// TIA Portal V20 export
DATA_BLOCK "ControlNodes"   // DB82
{ DB_Accessible_From_OPC_UA := 'FALSE' }
AUTHOR : ERsystem_FA2_DH. Kim
// stored: DBAccessibleFromOPCUA false, DBAccessibleFromWebserver false, MemoryReserve 100, Namespace Unit1.Em5
   VAR
      em { ExternalWritable := 'False'} : "LAF_typeEmControlNode";
      cm : Struct
         Interlock : Struct
            cathodeMainPnP1AxisX : "LER_typeAxisInterlock";
            cathodeMainPnP2AxisX : "LER_typeAxisInterlock";
            cathodeMainPnP1AxisY : "LER_typeAxisInterlock";
            cathodeMainPnP1AxisZ : "LER_typeAxisInterlock";
            cathodeMainPnP2AxisZ : "LER_typeAxisInterlock";
            cathodeAlignTableAxisX : "LER_typeAxisInterlock";
            cathodeAlignTableAxisY1 : "LER_typeAxisInterlock";
            cathodeAlignTableAxisY2 : "LER_typeAxisInterlock";
            cathodeMainPnP1RotaryCwCcw : "LER_typeTwoWayActInterlock";
            cathodeMainPnP1SuctionPlateVacuum : "LER_typeTwoWayActInterlock";
            cathodeMainPnP2SuctionPlateVacuum : "LER_typeTwoWayActInterlock";
            cathodeAlignTableSuctionPlateVacuum : "LER_typeTwoWayActInterlock";
            cathodeGlassCleaning : "LER_typeTwoWayActInterlock";
            cathodeNgPnpUpDown : "LER_typeTwoWayActInterlock";
            cathodeNgPnp1stFwdBwd : "LER_typeTwoWayActInterlock";
            cathodeNgPnp2ndFwdBwd : "LER_typeTwoWayActInterlock";
            cathodeMaintenanceMovingFixFwdBwd : "LER_typeTwoWayActInterlock";
            cathodeNgBoxLiftUpDown : "LER_typeTwoWayActInterlock";
            cathodeNgBoxLockUpDown : "LER_typeTwoWayActInterlock";
            cathodeNgPnpVaccum : "LER_typeTwoWayActInterlock";
            cathodeConveyorCoverFwdBwd : "LER_typeTwoWayActInterlock";
            cathodeConveyorPickUpBlower : "LER_typeTwoWayActInterlock";
         END_STRUCT;
         axisCommand : Struct
            cathodeMainPnP1AxisX : "LER_typeAxisCommand";
            cathodeMainPnP2AxisX : "LER_typeAxisCommand";
            cathodeMainPnP1AxisY : "LER_typeAxisCommand";
            cathodeMainPnP1AxisZ : "LER_typeAxisCommand";
            cathodeMainPnP2AxisZ : "LER_typeAxisCommand";
            cathodeAlignTableAxisX : "LER_typeAxisCommand";
            cathodeAlignTableAxisY1 : "LER_typeAxisCommand";
            cathodeAlignTableAxisY2 : "LER_typeAxisCommand";
         END_STRUCT;
         softCam : "Unit1.type_emRelations_em5_SoftCam";
         brakeTest : Struct
            cathodeMainPnP1AxisZ : "LER_typeBrakeTestEmControlNoeds";
            cathodeMainPnP2AxisZ : "LER_typeBrakeTestEmControlNoeds";
         END_STRUCT;
      END_STRUCT;
      mainPnP : Struct
         jobs : "LAF_typeJobs";
         sequence { S7_SetPoint := 'True'} : "LAF_typeSequence";
         "step" { S7_SetPoint := 'True'} : "LER_typeStep";
         jobInterface : Struct
            homeJob10 : "LER_typeJobInterface";
            homeJob1 : "LER_typeJobInterface";
            loadJob2 : "LER_typeJobInterface";
            unloadJob3 : "LER_typeJobInterface";
            avoidJob4 : "LER_typeJobInterface";
            oneLoadJob5 : "LER_typeJobInterface";
            oneUnLoadJob6 : "LER_typeJobInterface";
         END_STRUCT;
         preOperationCheck : Struct
            partNoDetect1 : Bool;   // MainPnP1/2 No Have Cell In LoadPos
            partNoDetect2 : Bool;
            partDetect1 : Bool;
            partDetect2 : Bool;
            partNG : Bool;
            Bool6 : Bool;
            Bool7 : Bool;
            Bool8 : Bool;   // MainPnP1 Have Cell
            Bool9 : Bool;   // MainPnP1/2 No Have Cell In UnLoadPos
            Bool10 : Bool;   // MainPnP1/2 Have Cell
            Bool11 : Bool;   // MainPnP1/2 Have Cell But Cathde Turn
            Bool12 : Bool;   // EM5 Ready For Motion
            Bool13 : Bool;
            Bool14 : Bool;
            Bool15 : Bool;
            Bool16 : Bool;
            Bool17 : Bool;
            Bool18 : Bool;
            Bool19 : Bool;
            Bool20 : Bool;
         END_STRUCT;
      END_STRUCT;
      alignTable : Struct
         jobs : "LAF_typeJobs";
         sequence { S7_SetPoint := 'True'} : "LAF_typeSequence";
         "step" { S7_SetPoint := 'True'} : "LER_typeStep";
         jobInterface : Struct
            homeJob1 : "LER_typeJobInterface";
            loadJob2 : "LER_typeJobInterface";
            visionJob3 : "LER_typeJobInterface";
            unloadJob4 : "LER_typeJobInterface";
         END_STRUCT;
         preOperationCheck : Struct
            partNoDetect1 : Bool;   // AlignTable No Have Cell In WaitPos
            partNoDetect2 : Bool;   // AlignTable No Have Cell In AdjustPos
            partDetect1 : Bool;   // AlignTable Have Cell In WaitPos
            partDetect2 : Bool;   // AlignTable Have Cell In AdjustPos
            Bool5 : Bool;
            Bool6 : Bool;
            Bool7 : Bool;
            Bool8 : Bool;
            Bool9 : Bool;
            Bool10 : Bool;
            Bool11 : Bool;
            Bool12 : Bool;
            Bool13 : Bool;
            Bool14 : Bool;
            Bool15 : Bool;
            Bool16 : Bool;
            Bool17 : Bool;
            Bool18 : Bool;
            Bool19 : Bool;
            Bool20 : Bool;
         END_STRUCT;
      END_STRUCT;
      ngPnP : Struct
         jobs : "LAF_typeJobs";
         sequence { S7_SetPoint := 'True'} : "LAF_typeSequence";
         "step" { S7_SetPoint := 'True'} : "LER_typeStep";
         jobInterface : Struct
            homeJob1 : "LER_typeJobInterface";
            loadJob2 : "LER_typeJobInterface";
            unloadJob3 : "LER_typeJobInterface";
         END_STRUCT;
         preOperationCheck : Struct
            partNoDetect : Bool;
            partDetect : Bool;
            Bool3 : Bool;
            Bool4 : Bool;
            Bool5 : Bool;
            Bool6 : Bool;
            Bool7 : Bool;
            Bool8 : Bool;
            Bool9 : Bool;
            Bool10 : Bool;
            Bool11 : Bool;
            Bool12 : Bool;
            Bool13 : Bool;
            Bool14 : Bool;
            Bool15 : Bool;
            Bool16 : Bool;
            Bool17 : Bool;
            Bool18 : Bool;
            Bool19 : Bool;
            Bool20 : Bool;
         END_STRUCT;
      END_STRUCT;
      gaugeRnR : Struct
         jobs : "LAF_typeJobs";
         sequence { S7_SetPoint := 'True'} : "LAF_typeSequence";
         "step" { S7_SetPoint := 'True'} : "LER_typeStep";
         jobInterface : Struct
            commonReadyJob1 : "LER_typeJobInterface";
            commonGetMasterPieceJob2 { S7_SetPoint := 'True'} : "LER_typeJobInterface";
            "1StackMainPnP2ToStackTableJob19" { S7_SetPoint := 'True'} : "LER_typeJobInterface";
            "1StackStackTableToMainPnP2Job20" { S7_SetPoint := 'True'} : "LER_typeJobInterface";
         END_STRUCT;
         homeCheck : Struct
            home : Bool;
         END_STRUCT;
      END_STRUCT;
      ReelCutInterface : Struct
         readyMasterPiece : Bool;
      END_STRUCT;
      emRelations : Struct
         em6 : Struct
            reqStackTableVaccum : Bool;
            reqStackTableBlow : Bool;
            readyGaugeRnR : Bool;
            doneStackTableVaccum : Bool;
            doneStackTableBlow : Bool;
            doneGaugeRnR : Bool;
            softCam : "Unit1.type_emRelations_em6_SoftCam";
         END_STRUCT;
      END_STRUCT;
      cmPnp1stCathodeDetect { S7_SetPoint := 'True'} : "LBC_typeDigitalSignalControlNode";
      cmPnp2ndCathodeDetect { S7_SetPoint := 'True'} : "LBC_typeDigitalSignalControlNode";
      cmCathodeAlignTableElectrodeDetect { S7_SetPoint := 'True'} : "LBC_typeDigitalSignalControlNode";
      cmCathodeNgPnpElectrodeDetect { S7_SetPoint := 'True'} : "LBC_typeDigitalSignalControlNode";
      cmCathodeNgBoxFullSensorDetect { S7_SetPoint := 'True'} : "LBC_typeDigitalSignalControlNode";
      cmCathodeNgBoxDetect { S7_SetPoint := 'True'} : "LBC_typeDigitalSignalControlNode";
      cmCathodeMainPnP1AxisX { ExternalAccessible := 'False'; ExternalVisible := 'False'; ExternalWritable := 'False'} : "LBC_typeAxis64PosControlNode";
      cmCathodeMainPnP2AxisX { ExternalAccessible := 'False'; ExternalVisible := 'False'; ExternalWritable := 'False'} : "LBC_typeAxis64PosControlNode";
      cmCathodeMainPnP1AxisY { ExternalAccessible := 'False'; ExternalVisible := 'False'; ExternalWritable := 'False'} : "LBC_typeAxis64PosControlNode";
      cmCathodeMainPnP1AxisZ { ExternalAccessible := 'False'; ExternalVisible := 'False'; ExternalWritable := 'False'} : "LBC_typeAxis64PosControlNode";
      cmCathodeMainPnP2AxisZ { ExternalAccessible := 'False'; ExternalVisible := 'False'; ExternalWritable := 'False'} : "LBC_typeAxis64PosControlNode";
      cmCathodeAlignTableAxisX { ExternalAccessible := 'False'; ExternalVisible := 'False'; ExternalWritable := 'False'} : "LBC_typeAxis64PosControlNode";
      cmCathodeAlignTableAxisY1 { ExternalAccessible := 'False'; ExternalVisible := 'False'; ExternalWritable := 'False'} : "LBC_typeAxis64PosControlNode";
      cmCathodeAlignTableAxisY2 { ExternalAccessible := 'False'; ExternalVisible := 'False'; ExternalWritable := 'False'} : "LBC_typeAxis64PosControlNode";
      cmCathodeMainPnP1RotaryCwCcw { ExternalAccessible := 'False'; ExternalVisible := 'False'; ExternalWritable := 'False'} : "LBC_typeTwoWayActuatorControlNode";
      cmCathodeMainPnP1SuctionPlateVacuum { ExternalAccessible := 'False'; ExternalVisible := 'False'; ExternalWritable := 'False'} : "LBC_typeTwoWayActuatorControlNode";
      cmCathodeMainPnP2SuctionPlateVacuum { ExternalAccessible := 'False'; ExternalVisible := 'False'; ExternalWritable := 'False'} : "LBC_typeTwoWayActuatorControlNode";
      cmCathodeAlignTableSuctionPlateVacuum { ExternalAccessible := 'False'; ExternalVisible := 'False'; ExternalWritable := 'False'} : "LBC_typeTwoWayActuatorControlNode";
      cmCathodeGlassCleaning { ExternalAccessible := 'False'; ExternalVisible := 'False'; ExternalWritable := 'False'} : "LBC_typeTwoWayActuatorControlNode";
      cmCathodeNgPnpUpDown { ExternalAccessible := 'False'; ExternalVisible := 'False'; ExternalWritable := 'False'} : "LBC_typeTwoWayActuatorControlNode";
      cmCathodeNgPnp1stFwdBwd { ExternalAccessible := 'False'; ExternalVisible := 'False'; ExternalWritable := 'False'} : "LBC_typeTwoWayActuatorControlNode";
      cmCathodeNgPnp2ndFwdBwd { ExternalAccessible := 'False'; ExternalVisible := 'False'; ExternalWritable := 'False'; S7_SetPoint := 'True'} : "LBC_typeTwoWayActuatorControlNode";
      cmCathodeMaintenanceMovingFixFwdBwd { ExternalAccessible := 'False'; ExternalVisible := 'False'; ExternalWritable := 'False'} : "LBC_typeTwoWayActuatorControlNode";
      cmCathodeNgBoxLiftUpDown { ExternalAccessible := 'False'; ExternalVisible := 'False'; ExternalWritable := 'False'; S7_SetPoint := 'True'} : "LBC_typeTwoWayActuatorControlNode";
      cmCathodeNgBoxLockUpDown { ExternalAccessible := 'False'; ExternalVisible := 'False'; ExternalWritable := 'False'; S7_SetPoint := 'True'} : "LBC_typeTwoWayActuatorControlNode";
      cmCathodeNgPnpVaccum { ExternalAccessible := 'False'; ExternalVisible := 'False'; ExternalWritable := 'False'} : "LBC_typeTwoWayActuatorControlNode";
      cmCathodeConveyorCoverFwdBwd { S7_SetPoint := 'True'} : "LBC_typeTwoWayActuatorControlNode";
      cmCathodeConveyorPickUpBlower { S7_SetPoint := 'True'} : "LBC_typeTwoWayActuatorControlNode";
      cmCathodeVisionControllerInterface { ExternalAccessible := 'False'; ExternalVisible := 'False'; ExternalWritable := 'False'} : "LER_typeVisionControlNode";
   END_VAR
BEGIN
   em.commands.enable := FALSE;
   em.commands.acknowledge := FALSE;
   em.commands.disableAlarms := FALSE;
   em.commands.activateSimulation := FALSE;
   em.commands.home := FALSE;
   em.commands.moveToInitialPosition := FALSE;
   em.commands.directModeControl.current := 2;
   em.commands.directModeControl.production := FALSE;
   em.commands.directModeControl.maintenance := TRUE;
   em.commands.directModeControl.manual := FALSE;
   em.commands.directModeControl.nomode := FALSE;
   em.commands.directModeControl.sleep := FALSE;
   em.commands.directModeControl.deepsleep := FALSE;
   em.commands.directModeControl.userMode04 := FALSE;
   em.commands.directModeControl.userMode05 := FALSE;
   em.commands.directModeControl.userMode06 := FALSE;
   em.commands.directModeControl.userMode07 := FALSE;
   em.commands.directModeControl.userMode08 := FALSE;
   em.commands.directModeControl.userMode09 := FALSE;
   em.commands.directModeControl.userMode10 := FALSE;
   em.commands.directModeControl.userMode11 := FALSE;
   em.commands.directModeControl.userMode12 := FALSE;
   em.commands.directModeControl.userMode13 := FALSE;
   em.commands.directStateControl.current := 2;
   em.commands.directStateControl.clearing := FALSE;
   em.commands.directStateControl.stopped := TRUE;
   em.commands.directStateControl.starting := FALSE;
   em.commands.directStateControl.idle := FALSE;
   em.commands.directStateControl.suspended := FALSE;
   em.commands.directStateControl.execute := FALSE;
   em.commands.directStateControl.stopping := FALSE;
   em.commands.directStateControl.aborting := FALSE;
   em.commands.directStateControl.aborted := FALSE;
   em.commands.directStateControl.holding := FALSE;
   em.commands.directStateControl.held := FALSE;
   em.commands.directStateControl.unholding := FALSE;
   em.commands.directStateControl.suspending := FALSE;
   em.commands.directStateControl.unsuspending := FALSE;
   em.commands.directStateControl.resetting := FALSE;
   em.commands.directStateControl.completing := FALSE;
   em.commands.directStateControl.complete := FALSE;
   em.status.enabled := FALSE;
   em.status.acknowledgeActive := FALSE;
   em.status.alarmsDisabled := FALSE;
   em.status.simulationActive := FALSE;
   em.status.safetyReleased := TRUE;
   em.status.initialized := FALSE;
   em.status.homed := TRUE;
   em.status.safeState := FALSE;
   em.status.stateComplete := TRUE;
   // mainPnP."step".action1[101] : Step[101] : JOB[1] Condition
   // mainPnP."step".action1[110] : Step[110] : Main P&P 1,2 Z-Axis Wait Pos
   // mainPnP."step".action1[111] : Step[111] : Main P&P 1 Y-Axis Wait Pos
   // mainPnP."step".action1[112] : Step[112] : Main P&P 1,2 X-Axis Wait(=Load) Pos
   // mainPnP."step".action1[113] : Step[113] : Main P&P 1 Rotary Cylinder InHomePos(=Clock Wise)
   // mainPnP."step".action1[114] : Step[114] : Main P&P 1 Z-Axis Load Pos
   // mainPnP."step".action1[115] : Step[115] : Main P&P 1 Vaccum On
   // mainPnP."step".action1[116] : Step[116] : Main P&P 1 Pick Up Blow On
   // mainPnP."step".action1[117] : Step[117] : Main P&P 1,2 Z-Axis Wait Pos
   // mainPnP."step".action1[120] : Step[120] : Main P&P 1,2 X-Axis Unload Pos
   // mainPnP."step".action1[121] : Step[121] : Main P&P 1 Rotary Cylinder InWorkPos(=Counter Clock Wise)
   // mainPnP."step".action1[122] : Step[122] : Main P&P 1 Z-Axis Unload Pos [Request Check]
   // mainPnP."step".action1[123] : Step[123] : Main P&P → Align Table [Vacuum On Request]
   // mainPnP."step".action1[124] : Step[124] : Main P&P 1 Vaccum Off
   // mainPnP."step".action1[125] : Step[125] : Main P&P 1,2 Z-Axis Wait Pos
   // mainPnP."step".action1[130] : Step[130] : Main P&P 1,2 X-Axis Load Pos
   // mainPnP."step".action1[131] : Step[131] : Main P&P 1 Rotary Cylinder InHomePos(=Clock Wise)
   // mainPnP."step".action1[132] : Step[132] : Main P&P 1,2 Z-Axis Load Pos [Request Check]
   // mainPnP."step".action1[133] : Step[133] : Main P&P 1,2 Vaccum On
   // mainPnP."step".action1[134] : Step[134] : Main P&P → Align Table [Vacuum Off Request] / Pick Up Blow On
   // mainPnP."step".action1[135] : Step[135] : Main P&P 1,2 Z-Axis Wait Pos
   // mainPnP."step".action1[140] : Step[140] : Main P&P 1,2 X-Axis Unload Pos
   // mainPnP."step".action1[141] : Step[141] : Main P&P 1 Rotary Cylinder InWorkPos(=Counter Clock Wise)
   // mainPnP."step".action1[142] : Step[142] : Main P&P 1,2 Z-Axis Unload Pos [Request Check]
   // mainPnP."step".action1[143] : Step[143] : Main P&P → Align Table [Vacuum On Request] / Mendrel [Clamp Request]
   // mainPnP."step".action1[144] : Step[144] : Main P&P 1,2 Vaccum Off
   // mainPnP."step".action1[145] : Step[145] : Main P&P 1,2 Z-Axis Wait Pos
   // mainPnP."step".action1[180] : Step[180] : Main P&P 1,2 X-Axis Load Pos
   // mainPnP."step".action1[181] : Step[181] : Main P&P 1 Rotary Cylinder InHomePos(=Clock Wise)
   // mainPnP."step".action1[182] : Step[182] : Main P&P 1,2 Z-Axis Load Pos [Request Check]
   // mainPnP."step".action1[183] : Step[183] : Main P&P 1,2 Vaccum On
   // mainPnP."step".action1[184] : Step[184] : Main P&P → Align Table [Vacuum Off Request] / Pick Up Blow On
   // mainPnP."step".action1[185] : Step[185] : Main P&P 1,2 Z-Axis Avoid Pos
   // mainPnP."step".action1[190] : Step[190] : JOB[1] Step End
   // mainPnP."step".action1[201] : Step[201] : JOB[2] Condition
   // mainPnP."step".action1[210] : Step[210] : Main P&P 1,2 Z-Axis Wait Pos
   // mainPnP."step".action1[220] : Step[220] : Main P&P 1,2 X-Axis Load Pos
   // mainPnP."step".action1[230] : Step[230] : Main P&P 1 Rotary Cylinder InHomePos(=Clock Wise)
   // mainPnP."step".action1[240] : Step[240] : Main P&P 1.2 Z-Axis Load Pos
   // mainPnP."step".action1[250] : Step[250] : Main P&P 1,2 Vaccum On
   // mainPnP."step".action1[260] : Step[260] : Main P&P → Align Table [Vacuum Off Request] / Pick Up Blow On
   // mainPnP."step".action1[280] : Step[280] : Main P&P 1,2 Z-Axis Wait Pos
   // mainPnP."step".action1[290] : Step[290] : JOB[2] Condition
   // mainPnP."step".action1[301] : Step[301] : JOB[3] Condition
   // mainPnP."step".action1[310] : Step[310] : Main P&P 1,2 Z-Axis Wait Pos
   // mainPnP."step".action1[320] : Step[320] : Main P&P 1,2 X-Axis Unload Pos
   // mainPnP."step".action1[330] : Step[330] : Main P&P 1 Rotary Cylinder InWorkPos(=Counter Clock Wise)
   // mainPnP."step".action1[340] : Step[340] : Main P&P 1.2 Z-Axis Unload Pos
   // mainPnP."step".action1[350] : Step[350] : Main P&P → Align Table [Vacuum On Request] / Mendrel [Clamp Request]
   // mainPnP."step".action1[360] : Step[360] : Main P&P 1.2 Vaccum Off
   // mainPnP."step".action1[380] : Step[380] : Main P&P 1,2 Z-Axis Wait Pos
   // mainPnP."step".action1[390] : Step[390] : JOB[3] Condition
   // mainPnP."step".action1[401] : Step[401] : JOB[4] Condition
   // mainPnP."step".action1[420] : Step[420] : Main P&P 1 X-Axis Load Pos, Main P&P 2 X-Axis Unload Pos
   // mainPnP."step".action1[430] : Step[430] : Main P&P 1 Rotary Cylinder InHomePos(=Clock Wise)
   // mainPnP."step".action1[490] : Step[490] : JOB[3] Condition
   // mainPnP."step".transition1[101] : Step[101] : JOB[1] Condition
   // mainPnP."step".transition1[110] : Step[110] : Main P&P 1,2 Z-Axis Wait Pos
   // mainPnP."step".transition1[111] : Step[111] : Main P&P 1 Y-Axis Wait Pos
   // mainPnP."step".transition1[112] : Step[112] : Main P&P 1,2 X-Axis Wait(=Load) Pos
   // mainPnP."step".transition1[113] : Step[113] : Main P&P 1 Rotary Cylinder InHomePos(=Clock Wise)
   // mainPnP."step".transition1[114] : Step[114] : Main P&P 1 Z-Axis Load Pos
   // mainPnP."step".transition1[115] : Step[115] : Main P&P 1 Vaccum On
   // mainPnP."step".transition1[116] : Step[116] : Main P&P 1 Pick Up Blow On
   // mainPnP."step".transition1[117] : Step[117] : Main P&P 1,2 Z-Axis Wait Pos
   // mainPnP."step".transition1[120] : Step[120] : Main P&P 1,2 X-Axis Unload Pos
   // mainPnP."step".transition1[121] : Step[121] : Main P&P 1 Rotary Cylinder InWorkPos(=Counter Clock Wise)
   // mainPnP."step".transition1[122] : Step[122] : Main P&P 1 Z-Axis Unload Pos [Request Check]
   // mainPnP."step".transition1[123] : Step[123] : Main P&P → Align Table [Vacuum On Request]
   // mainPnP."step".transition1[124] : Step[124] : Main P&P 1 Vaccum Off
   // mainPnP."step".transition1[125] : Step[125] : Main P&P 1,2 Z-Axis Wait Pos
   // mainPnP."step".transition1[130] : Step[130] : Main P&P 1,2 X-Axis Load Pos
   // mainPnP."step".transition1[131] : Step[131] : Main P&P 1 Rotary Cylinder InHomePos(=Clock Wise)
   // mainPnP."step".transition1[132] : Step[132] : Main P&P 1,2 Z-Axis Load Pos [Request Check]
   // mainPnP."step".transition1[133] : Step[133] : Main P&P 1,2 Vaccum On
   // mainPnP."step".transition1[134] : Step[134] : Main P&P → Align Table [Vacuum Off Request] / Pick Up Blow On
   // mainPnP."step".transition1[135] : Step[135] : Main P&P 1,2 Z-Axis Wait Pos
   // mainPnP."step".transition1[140] : Step[140] : Main P&P 1,2 X-Axis Unload Pos
   // mainPnP."step".transition1[141] : Step[141] : Main P&P 1 Rotary Cylinder InWorkPos(=Counter Clock Wise)
   // mainPnP."step".transition1[142] : Step[142] : Main P&P 1,2 Z-Axis Unload Pos [Request Check]
   // mainPnP."step".transition1[143] : Step[143] : Main P&P → Align Table [Vacuum On Request] / Mendrel [Clamp Request]
   // mainPnP."step".transition1[144] : Step[144] : Main P&P 1,2 Vaccum Off
   // mainPnP."step".transition1[145] : Step[145] : Main P&P 1,2 Z-Axis Wait Pos
   // mainPnP."step".transition1[180] : Step[180] : Main P&P 1,2 X-Axis Load Pos
   // mainPnP."step".transition1[181] : Step[181] : Main P&P 1 Rotary Cylinder InHomePos(=Clock Wise)
   // mainPnP."step".transition1[182] : Step[182] : Main P&P 1,2 Z-Axis Load Pos [Request Check]
   // mainPnP."step".transition1[183] : Step[183] : Main P&P 1,2 Vaccum On
   // mainPnP."step".transition1[184] : Step[184] : Main P&P → Align Table [Vacuum Off Request] / Pick Up Blow On
   // mainPnP."step".transition1[185] : Step[185] : Main P&P 1,2 Z-Axis Avoid Pos
   // mainPnP."step".transition1[190] : Step[190] : JOB[1] Step End
   // mainPnP."step".transition1[201] : Step[201] : JOB[2] Condition
   // mainPnP."step".transition1[210] : Step[210] : Main P&P 1,2 Z-Axis Wait Pos
   // mainPnP."step".transition1[220] : Step[220] : Main P&P 1,2 X-Axis Load Pos
   // mainPnP."step".transition1[230] : Step[230] : Main P&P 1 Rotary Cylinder InHomePos(=Clock Wise)
   // mainPnP."step".transition1[240] : Step[240] : Main P&P 1.2 Z-Axis Load Pos
   // mainPnP."step".transition1[250] : Step[250] : Main P&P 1,2 Vaccum On
   // mainPnP."step".transition1[260] : Step[260] : Main P&P → Align Table [Vacuum Off Request] / Pick Up Blow On
   // mainPnP."step".transition1[280] : Step[280] : Main P&P 1,2 Z-Axis Wait Pos
   // mainPnP."step".transition1[290] : Step[290] : JOB[2] Condition
   // mainPnP."step".transition1[301] : Step[301] : JOB[3] Condition
   // mainPnP."step".transition1[310] : Step[310] : Main P&P 1,2 Z-Axis Wait Pos
   // mainPnP."step".transition1[320] : Step[320] : Main P&P 1,2 X-Axis Unload Pos
   // mainPnP."step".transition1[330] : Step[330] : Main P&P 1 Rotary Cylinder InWorkPos(=Counter Clock Wise)
   // mainPnP."step".transition1[340] : Step[340] : Main P&P 1.2 Z-Axis Unload Pos
   // mainPnP."step".transition1[350] : Step[350] : Main P&P → Align Table [Vacuum On Request] / Mendrel [Clamp Request]
   // mainPnP."step".transition1[360] : Step[360] : Main P&P 1.2 Vaccum Off
   // mainPnP."step".transition1[380] : Step[380] : Main P&P 1,2 Z-Axis Wait Pos
   // mainPnP."step".transition1[390] : Step[390] : JOB[3] Condition
   // mainPnP."step".transition1[401] : Step[401] : JOB[4] Condition
   // mainPnP."step".transition1[420] : Step[420] : Main P&P 1 X-Axis Load Pos, Main P&P 2 X-Axis Unload Pos
   // mainPnP."step".transition1[430] : Step[430] : Main P&P 1 Rotary Cylinder InHomePos(=Clock Wise)
   // mainPnP."step".transition1[490] : Step[490] : JOB[3] Condition
   // alignTable."step".action1[101] : Step[101] : JOB[1] Condition
   // alignTable."step".action1[110] : Step[110] : Vaccum Off
   // alignTable."step".action1[120] : Step[120] : Glass Cleaning On [Main P&P Working Done Check]
   // alignTable."step".action1[140] : Step[140] : Align Table → Main P&P [Load Request]
   // alignTable."step".action1[141] : Step[141] : Vaccum On
   // alignTable."step".action1[142] : Step[142] : Align Table → Main P&P [Load Done] / [Vision Unuse Check]
   // alignTable."step".action1[150] : Step[150] : Vision Start
   // alignTable."step".action1[151] : Step[151] : Vision Result
   // alignTable."step".action1[152] : Step[152] : Align Table X,Y1,Y2-Axis Work Pos
   // alignTable."step".action1[160] : Step[160] : Align Table → Main P&P/NG P&P [Unload Request]
   // alignTable."step".action1[161] : Step[161] : Vaccum Off
   // alignTable."step".action1[162] : Step[162] : Align Table → Main P&P [Unload Done]
   // alignTable."step".action1[163] : Step[163] : Glass Cleaning On [Main P&P Homing Job Complete Check]
   // alignTable."step".action1[180] : Step[180] : Align Table X,Y1,Y2-Axis Wait Pos
   // alignTable."step".action1[190] : Step[190] : JOB[1] Step End
   // alignTable."step".action1[201] : Step[201] : JOB[2] Condition
   // alignTable."step".action1[210] : Step[210] : Align Table → Main P&P [Load Request]
   // alignTable."step".action1[220] : Step[220] : Vaccum On
   // alignTable."step".action1[230] : Step[230] : Align Table → Main P&P [Load Done]
   // alignTable."step".action1[290] : Step[290] : JOB[2] Condition
   // alignTable."step".action1[301] : Step[301] : JOB[3] Condition
   // alignTable."step".action1[310] : Step[310] : Vision Start
   // alignTable."step".action1[320] : Step[320] : Vision Result
   // alignTable."step".action1[380] : Step[380] : Align Table X,Y1,Y2-Axis Work Pos
   // alignTable."step".action1[390] : Step[390] : JOB[3] Condition
   // alignTable."step".action1[401] : Step[401] : JOB[4] Condition
   // alignTable."step".action1[410] : Step[410] : Align Table → Main P&P/NG P&P [Unload Request]
   // alignTable."step".action1[420] : Step[420] : Vaccum Off
   // alignTable."step".action1[430] : Step[430] : Align Table → Main P&P [Unload Done]
   // alignTable."step".action1[431] : Step[431] : Glass Cleaning On
   // alignTable."step".action1[480] : Step[480] : Align Table X,Y1,Y2-Axis Wait Pos
   // alignTable."step".transition1[101] : Step[101] : JOB[1] Condition
   // alignTable."step".transition1[110] : Step[110] : Vaccum Off
   // alignTable."step".transition1[120] : Step[120] : Glass Cleaning On [Main P&P Working Done Check]
   // alignTable."step".transition1[140] : Step[140] : Align Table → Main P&P [Load Request]
   // alignTable."step".transition1[141] : Step[141] : Vaccum On
   // alignTable."step".transition1[142] : Step[142] : Align Table → Main P&P [Load Done] / [Vision Unuse Check]
   // alignTable."step".transition1[150] : Step[150] : Vision Start
   // alignTable."step".transition1[151] : Step[151] : Vision Result
   // alignTable."step".transition1[152] : Step[152] : Align Table X,Y1,Y2-Axis Work Pos
   // alignTable."step".transition1[160] : Step[160] : Align Table → Main P&P/NG P&P [Unload Request]
   // alignTable."step".transition1[161] : Step[161] : Vaccum Off
   // alignTable."step".transition1[162] : Step[162] : Align Table → Main P&P [Unload Done]
   // alignTable."step".transition1[163] : Step[163] : Glass Cleaning On [Main P&P Homing Job Complete Check]
   // alignTable."step".transition1[180] : Step[180] : Align Table X,Y1,Y2-Axis Wait Pos
   // alignTable."step".transition1[190] : Step[190] : JOB[1] Step End
   // alignTable."step".transition1[201] : Step[201] : JOB[2] Condition
   // alignTable."step".transition1[210] : Step[210] : Align Table → Main P&P [Load Request]
   // alignTable."step".transition1[220] : Step[220] : Vaccum On
   // alignTable."step".transition1[230] : Step[230] : Align Table → Main P&P [Load Done]
   // alignTable."step".transition1[290] : Step[290] : JOB[2] Condition
   // alignTable."step".transition1[301] : Step[301] : JOB[3] Condition
   // alignTable."step".transition1[310] : Step[310] : Vision Start
   // alignTable."step".transition1[320] : Step[320] : Vision Result
   // alignTable."step".transition1[380] : Step[380] : Align Table X,Y1,Y2-Axis Work Pos
   // alignTable."step".transition1[390] : Step[390] : JOB[3] Condition
   // alignTable."step".transition1[401] : Step[401] : JOB[4] Condition
   // alignTable."step".transition1[410] : Step[410] : Align Table → Main P&P/NG P&P [Unload Request]
   // alignTable."step".transition1[420] : Step[420] : Vaccum Off
   // alignTable."step".transition1[430] : Step[430] : Align Table → Main P&P [Unload Done]
   // alignTable."step".transition1[431] : Step[431] : Glass Cleaning On
   // alignTable."step".transition1[480] : Step[480] : Align Table X,Y1,Y2-Axis Wait Pos
   // ngPnP."step".action1[101] : Step[101] : JOB[1] Condition
   // ngPnP."step".action1[110] : Step[110] : Vaccum Off
   // ngPnP."step".action1[120] : Step[120] : NG P&P Up
   // ngPnP."step".action1[130] : Step[130] : NG P&P 1,2 Backward
   // ngPnP."step".action1[180] : Step[180] : Lift Down
   // ngPnP."step".action1[190] : Step[190] : JOB[1] Step End
   // ngPnP."step".action1[201] : Step[201] : JOB[2] Condition
   // ngPnP."step".action1[210] : Step[210] : NG P&P 1,2 Forward
   // ngPnP."step".action1[220] : Step[220] : NG P&P Down
   // ngPnP."step".action1[230] : Step[230] : Vaccum On
   // ngPnP."step".action1[231] : Step[231] : NG P&P → Align Table [Loading Ready]
   // ngPnP."step".action1[240] : Step[240] : NG P&P Up
   // ngPnP."step".action1[280] : Step[280] : NG P&P 1,2 Backward
   // ngPnP."step".action1[290] : Step[290] : JOB[2] Condition
   // ngPnP."step".action1[301] : Step[301] : JOB[3] Condition
   // ngPnP."step".action1[320] : Step[320] : NG P&P Down
   // ngPnP."step".action1[330] : Step[330] : Vaccum Off
   // ngPnP."step".action1[340] : Step[340] : NG P&P Up
   // ngPnP."step".action1[390] : Step[390] : JOB[3] Condition
   // ngPnP."step".transition1[101] : Step[101] : JOB[1] Condition
   // ngPnP."step".transition1[110] : Step[110] : Vaccum Off
   // ngPnP."step".transition1[120] : Step[120] : NG P&P Up
   // ngPnP."step".transition1[130] : Step[130] : NG P&P 1,2 Backward
   // ngPnP."step".transition1[180] : Step[180] : Lift Down
   // ngPnP."step".transition1[190] : Step[190] : JOB[1] Step End
   // ngPnP."step".transition1[201] : Step[201] : JOB[2] Condition
   // ngPnP."step".transition1[210] : Step[210] : NG P&P 1,2 Forward
   // ngPnP."step".transition1[220] : Step[220] : NG P&P Down
   // ngPnP."step".transition1[230] : Step[230] : Vaccum On
   // ngPnP."step".transition1[231] : Step[231] : NG P&P → Align Table [Loading Ready]
   // ngPnP."step".transition1[240] : Step[240] : NG P&P Up
   // ngPnP."step".transition1[280] : Step[280] : NG P&P 1,2 Backward
   // ngPnP."step".transition1[290] : Step[290] : JOB[2] Condition
   // ngPnP."step".transition1[301] : Step[301] : JOB[3] Condition
   // ngPnP."step".transition1[320] : Step[320] : NG P&P Down
   // ngPnP."step".transition1[330] : Step[330] : Vaccum Off
   // ngPnP."step".transition1[340] : Step[340] : NG P&P Up
   // ngPnP."step".transition1[390] : Step[390] : JOB[3] Condition
   // gaugeRnR."step".action1[101] : Step[101] : JOB[1] Condition
   // gaugeRnR."step".action1[110] : Step[110] : MainPnP 1 Vaccum Off
   // gaugeRnR."step".action1[120] : Step[120] : MainPnP 2 Vaccum Off
   // gaugeRnR."step".action1[130] : Step[130] : AlignTable Vaccum Off
   // gaugeRnR."step".action1[190] : Step[190] : Job[1] Step End
   // gaugeRnR."step".action1[201] : Step[201] : JOB[2] Condition
   // gaugeRnR."step".action1[210] : Step[210] : MainPnP1 Z-Axis Conveyor Down
   // gaugeRnR."step".action1[220] : Step[220] : MainPnP1 C/V Blow On
   // gaugeRnR."step".action1[230] : Step[230] : MainPnP1 Vaccum On
   // gaugeRnR."step".action1[240] : Step[240] : MainPnP1 C/V Blow Off
   // gaugeRnR."step".action1[250] : Step[250] : MainPnP1 Z-Axis Up
   // gaugeRnR."step".action1[290] : Step[290] : Job[2] Step End
   // gaugeRnR."step".action1[301] : Step[301] : JOB[3] Condition
   // gaugeRnR."step".action1[310] : Step[310] : MainPnP2 X-Axis Move StackTable
   // gaugeRnR."step".action1[320] : Step[320] : MainPnP1 X-Axis Move AlignTable
   // gaugeRnR."step".action1[390] : Step[390] : Job[3] Step End
   // gaugeRnR."step".action1[401] : Step[401] : Job[4] Condtion
   // gaugeRnR."step".action1[410] : Step[410] : MainPnP1 Z-Axis Down AlginTable
   // gaugeRnR."step".action1[420] : Step[420] : MainPnP1 1 Vaccum Off
   // gaugeRnR."step".action1[430] : Step[430] : AlignTable Vaccum On
   // gaugeRnR."step".action1[440] : Step[440] : MainPnP 1 Z-Axis Up
   // gaugeRnR."step".action1[490] : Step[490] : Job[4] Step End
   // gaugeRnR."step".action1[501] : Step[501] : Job[5] Condtion
   // gaugeRnR."step".action1[510] : Step[510] : MainPnP1 X-Axis Move ReelCut Convyeor
   // gaugeRnR."step".action1[520] : Step[520] : MainPnP2 X-Axis Move AlignTable
   // gaugeRnR."step".action1[590] : Step[590] : Job[5] Step End
   // gaugeRnR."step".action1[601] : Step[601] : Job[6] Condtion
   // gaugeRnR."step".action1[610] : Step[610] : AlignTable Vision Trigger On
   // gaugeRnR."step".action1[620] : Step[620] : AlignTable Move Adjust Pos
   // gaugeRnR."step".action1[690] : Step[690] : Job[6] Step End
   // gaugeRnR."step".action1[701] : Step[701] : Job[7] Condtion
   // gaugeRnR."step".action1[710] : Step[710] : MainPnP2 Z-Axis Down AlignTagble
   // gaugeRnR."step".action1[720] : Step[720] : AlignTable Vaccum Off
   // gaugeRnR."step".action1[730] : Step[730] : MainPnP2 Vaccum On
   // gaugeRnR."step".action1[740] : Step[740] : MainPnP2 Z-Axis Up
   // gaugeRnR."step".action1[790] : Step[790] : Job[7] Step End
   // gaugeRnR."step".action1[801] : Step[801] : Job[8] Condtion
   // gaugeRnR."step".action1[810] : Step[810] : AlignTable Move Wait
   // gaugeRnR."step".action1[890] : Step[890] : Job[8] Step End
   // gaugeRnR."step".action1[901] : Step[901] : Job[9] Condtion
   // gaugeRnR."step".action1[910] : Step[910] : MainPnP2 X-Axis Move StackTable
   // gaugeRnR."step".action1[990] : Step[990] : Job[9] Step End
   // gaugeRnR."step".action1[1001] : Step[1001] : Job[10] Condtion
   // gaugeRnR."step".action1[1010] : Step[1010] : MainPnP2 Z-Axis Move StackTable Down
   // gaugeRnR."step".action1[1020] : Step[1020] : MainPnP2 Vaccum Off
   // gaugeRnR."step".action1[1030] : Step[1030] : StackTable Vaccum On
   // gaugeRnR."step".action1[1040] : Step[1040] : MainPnP2 Z-Axis Up
   // gaugeRnR."step".action1[1090] : Step[1090] : Job[10] Step End
   // gaugeRnR."step".action1[1101] : Step[1101] : Job[11] Condtion
   // gaugeRnR."step".action1[1110] : Step[1110] : MainPnP2 Z-Axis Move StackTable Down
   // gaugeRnR."step".action1[1120] : Step[1120] : StackTable Vaccum Off
   // gaugeRnR."step".action1[1130] : Step[1130] : MainPnP2 Vaccum On
   // gaugeRnR."step".action1[1140] : Step[1140] : MainPnP2 Z-axis Up
   // gaugeRnR."step".action1[1190] : Step[1190] Job[11] Step End
   // gaugeRnR."step".action1[1201] : Step[1201] : Job[12] Condtion
   // gaugeRnR."step".action1[1210] : Step[1210] : MainPnP2 X-Axis Move AlignTable
   // gaugeRnR."step".action1[1290] : Step[1290] : Job[12] Step End
   // gaugeRnR."step".action1[1301] : Step[1301] : Job[13] Condtion
   // gaugeRnR."step".action1[1310] : Step[1310] : MainPnP2 Z-Axis Move StackTable Down
   // gaugeRnR."step".action1[1315] : Step[1315] : StackTable Vaccum Off
   // gaugeRnR."step".action1[1320] : Step[1320] : MainPnP2 Vaccum On
   // gaugeRnR."step".action1[1325] : Step[1325] : MainPnP2 Z-Axis Up
   // gaugeRnR."step".action1[1328] : Step[1328] : MainPnP2 X-Axis Move AlignTable
   // gaugeRnR."step".action1[1330] : Step[1330] : MainPnP2 Z-Axis Down AlignTagble
   // gaugeRnR."step".action1[1335] : Step[1335] : MainPnP2 Vaccum Off
   // gaugeRnR."step".action1[1340] : Step[1340] : AlignTable Vaccum On
   // gaugeRnR."step".action1[1345] : Step[1345] : MainPnP2 Z-Axis Up
   // gaugeRnR."step".action1[1350] : Step[1350] : MainPnP2 X-Axis Move StackTable
   // gaugeRnR."step".action1[1390] : Step[1390] : Job[13] Step End
   // gaugeRnR."step".action1[1401] : Step[1401] : Job[14] Condtion
   // gaugeRnR."step".action1[1410] : Step[1410] : NgPnP Up
   // gaugeRnR."step".action1[1415] : Step[1415] : NgPnP 1st Forward
   // gaugeRnR."step".action1[1420] : Step[1420] : NgPnP 2nd Forward
   // gaugeRnR."step".action1[1425] : Step[1425] : NgPnP Down
   // gaugeRnR."step".action1[1430] : Step[1430] : AlignTable Vacuum Off
   // gaugeRnR."step".action1[1435] : Step[1435] : NgPnP Vaccum On
   // gaugeRnR."step".action1[1440] : Step[1440] : NgPnP Up
   // gaugeRnR."step".action1[1445] : Step[1445] : NgPnP 1st Backward
   // gaugeRnR."step".action1[1450] : Step[1450] : NgPnP 2nd Backward
   // gaugeRnR."step".action1[1455] : Step[1455] : NgPnp Down
   // gaugeRnR."step".action1[1460] : Step[1460] : NgPnP Vaccum Off
   // gaugeRnR."step".action1[1465] : Step[1465] : NgPnP Up
   // gaugeRnR."step".action1[1470] : Step[1470] : MainPnP2 X-Axis Move AlignTable
   // gaugeRnR."step".action1[1490] : Step[1490] : Job[14] Step End
   // gaugeRnR."step".transition1[101] : Step[101] : JOB[1] Condition
   // gaugeRnR."step".transition1[110] : Step[110] : MainPnP 1 Vaccum Off
   // gaugeRnR."step".transition1[120] : Step[120] : MainPnP 2 Vaccum Off
   // gaugeRnR."step".transition1[130] : Step[130] : AlignTable Vaccum Off
   // gaugeRnR."step".transition1[190] : Step[190] : Job[1] Step End
   // gaugeRnR."step".transition1[201] : Step[201] : JOB[2] Condition
   // gaugeRnR."step".transition1[210] : Step[210] : MainPnP1 Z-Axis Conveyor Down
   // gaugeRnR."step".transition1[220] : Step[220] : MainPnP1 C/V Blow On
   // gaugeRnR."step".transition1[230] : Step[230] : MainPnP1 Vaccum On
   // gaugeRnR."step".transition1[240] : Step[240] : MainPnP1 C/V Blow Off
   // gaugeRnR."step".transition1[250] : Step[250] : MainPnP1 Z-Axis Up
   // gaugeRnR."step".transition1[290] : Step[290] : Job[2] Step End
   // gaugeRnR."step".transition1[301] : Step[301] : JOB[3] Condition
   // gaugeRnR."step".transition1[310] : Step[310] : MainPnP2 X-Axis Move StackTable
   // gaugeRnR."step".transition1[320] : Step[320] : MainPnP1 X-Axis Move AlignTable
   // gaugeRnR."step".transition1[390] : Step[390] : Job[3] Step End
   // gaugeRnR."step".transition1[401] : Step[401] : Job[4] Condtion
   // gaugeRnR."step".transition1[410] : Step[410] : MainPnP1 Z-Axis Down AlginTable
   // gaugeRnR."step".transition1[420] : Step[420] : MainPnP1 1 Vaccum Off
   // gaugeRnR."step".transition1[430] : Step[430] : AlignTable Vaccum On
   // gaugeRnR."step".transition1[440] : Step[440] : MainPnP 1 Z-Axis Up
   // gaugeRnR."step".transition1[490] : Step[490] : Job[4] Step End
   // gaugeRnR."step".transition1[501] : Step[501] : Job[5] Condtion
   // gaugeRnR."step".transition1[510] : Step[510] : MainPnP1 X-Axis Move ReelCut Convyeor
   // gaugeRnR."step".transition1[520] : Step[520] : MainPnP2 X-Axis Move AlignTable
   // gaugeRnR."step".transition1[590] : Step[590] : Job[5] Step End
   // gaugeRnR."step".transition1[601] : Step[601] : Job[6] Condtion
   // gaugeRnR."step".transition1[610] : Step[610] : AlignTable Vision Trigger On
   // gaugeRnR."step".transition1[620] : Step[620] : AlignTable Move Adjust Pos
   // gaugeRnR."step".transition1[690] : Step[690] : Job[6] Step End
   // gaugeRnR."step".transition1[701] : Step[701] : Job[7] Condtion
   // gaugeRnR."step".transition1[710] : Step[710] : MainPnP2 Z-Axis Down AlignTagble
   // gaugeRnR."step".transition1[720] : Step[720] : AlignTable Vaccum Off
   // gaugeRnR."step".transition1[730] : Step[730] : MainPnP2 Vaccum On
   // gaugeRnR."step".transition1[740] : Step[740] : MainPnP2 Z-Axis Up
   // gaugeRnR."step".transition1[790] : Step[790] : Job[7] Step End
   // gaugeRnR."step".transition1[801] : Step[801] : Job[8] Condtion
   // gaugeRnR."step".transition1[810] : Step[810] : AlignTable Move Wait
   // gaugeRnR."step".transition1[890] : Step[890] : Job[8] Step End
   // gaugeRnR."step".transition1[901] : Step[901] : Job[9] Condtion
   // gaugeRnR."step".transition1[910] : Step[910] : MainPnP2 X-Axis Move StackTable
   // gaugeRnR."step".transition1[990] : Step[990] : Job[9] Step End
   // gaugeRnR."step".transition1[1001] : Step[1001] : Job[10] Condtion
   // gaugeRnR."step".transition1[1010] : Step[1010] : MainPnP2 Z-Axis Move StackTable Down
   // gaugeRnR."step".transition1[1020] : Step[1020] : MainPnP2 Vaccum Off
   // gaugeRnR."step".transition1[1030] : Step[1030] : StackTable Vaccum On
   // gaugeRnR."step".transition1[1040] : Step[1040] : MainPnP2 Z-Axis Up
   // gaugeRnR."step".transition1[1090] : Step[1090] : Job[10] Step End
   // gaugeRnR."step".transition1[1101] : Step[1101] : Job[11] Condtion
   // gaugeRnR."step".transition1[1110] : Step[1110] : MainPnP2 Z-Axis Move StackTable Down
   // gaugeRnR."step".transition1[1120] : Step[1120] : StackTable Vaccum Off
   // gaugeRnR."step".transition1[1130] : Step[1130] : MainPnP2 Vaccum On
   // gaugeRnR."step".transition1[1140] : Step[1140] : MainPnP2 Z-axis Up
   // gaugeRnR."step".transition1[1190] : Step[1190] Job[11] Step End
   // gaugeRnR."step".transition1[1201] : Step[1201] : Job[12] Condtion
   // gaugeRnR."step".transition1[1210] : Step[1210] : MainPnP2 X-Axis Move AlignTable
   // gaugeRnR."step".transition1[1290] : Step[1290] : Job[12] Step End
   // gaugeRnR."step".transition1[1301] : Step[1301] : Job[13] Condtion
   // gaugeRnR."step".transition1[1310] : Step[1310] : MainPnP2 Z-Axis Move StackTable Down
   // gaugeRnR."step".transition1[1315] : Step[1315] : StackTable Vaccum Off
   // gaugeRnR."step".transition1[1320] : Step[1320] : MainPnP2 Vaccum On
   // gaugeRnR."step".transition1[1325] : Step[1325] : MainPnP2 Z-Axis Up
   // gaugeRnR."step".transition1[1328] : Step[1328] : MainPnP2 X-Axis Move AlignTable
   // gaugeRnR."step".transition1[1330] : Step[1330] : MainPnP2 Z-Axis Down AlignTagble
   // gaugeRnR."step".transition1[1335] : Step[1335] : MainPnP2 Vaccum Off
   // gaugeRnR."step".transition1[1340] : Step[1340] : AlignTable Vaccum On
   // gaugeRnR."step".transition1[1345] : Step[1345] : MainPnP2 Z-Axis Up
   // gaugeRnR."step".transition1[1350] : Step[1350] : MainPnP2 X-Axis Move StackTable
   // gaugeRnR."step".transition1[1390] : Step[1390] : Job[13] Step End
   // gaugeRnR."step".transition1[1401] : Step[1401] : Job[14] Condtion
   // gaugeRnR."step".transition1[1410] : Step[1410] : NgPnP Up
   // gaugeRnR."step".transition1[1415] : Step[1415] : NgPnP 1st Forward
   // gaugeRnR."step".transition1[1420] : Step[1420] : NgPnP 2nd Forward
   // gaugeRnR."step".transition1[1425] : Step[1425] : NgPnP Down
   // gaugeRnR."step".transition1[1430] : Step[1430] : AlignTable Vacuum Off
   // gaugeRnR."step".transition1[1435] : Step[1435] : NgPnP Vaccum On
   // gaugeRnR."step".transition1[1440] : Step[1440] : NgPnP Up
   // gaugeRnR."step".transition1[1445] : Step[1445] : NgPnP 1st Backward
   // gaugeRnR."step".transition1[1450] : Step[1450] : NgPnP 2nd Backward
   // gaugeRnR."step".transition1[1455] : Step[1455] : NgPnp Down
   // gaugeRnR."step".transition1[1460] : Step[1460] : NgPnP Vaccum Off
   // gaugeRnR."step".transition1[1465] : Step[1465] : NgPnP Up
   // gaugeRnR."step".transition1[1470] : Step[1470] : MainPnP2 X-Axis Move AlignTable
   // gaugeRnR."step".transition1[1490] : Step[1490] : Job[14] Step End
   cmPnp1stCathodeDetect.commands.reset := FALSE;
   cmPnp1stCathodeDetect.commands.simulation := FALSE;
   cmPnp1stCathodeDetect.commands.quality := TRUE;
   cmPnp1stCathodeDetect.monitoring.valid := TRUE;
   cmPnp1stCathodeDetect.monitoring.busy := TRUE;
   cmPnp1stCathodeDetect.monitoring.error := FALSE;
   cmPnp1stCathodeDetect.monitoring.status := 16#0000;
   cmPnp1stCathodeDetect.monitoring.risingEdge := FALSE;
   cmPnp1stCathodeDetect.monitoring.fallingEdge := FALSE;
   cmPnp1stCathodeDetect.monitoring.processValue := FALSE;
   cmPnp2ndCathodeDetect.commands.reset := FALSE;
   cmPnp2ndCathodeDetect.commands.simulation := FALSE;
   cmPnp2ndCathodeDetect.commands.quality := TRUE;
   cmPnp2ndCathodeDetect.monitoring.valid := TRUE;
   cmPnp2ndCathodeDetect.monitoring.busy := TRUE;
   cmPnp2ndCathodeDetect.monitoring.error := FALSE;
   cmPnp2ndCathodeDetect.monitoring.status := 16#0000;
   cmPnp2ndCathodeDetect.monitoring.risingEdge := FALSE;
   cmPnp2ndCathodeDetect.monitoring.fallingEdge := FALSE;
   cmPnp2ndCathodeDetect.monitoring.processValue := FALSE;
   cmCathodeAlignTableElectrodeDetect.commands.reset := FALSE;
   cmCathodeAlignTableElectrodeDetect.commands.simulation := FALSE;
   cmCathodeAlignTableElectrodeDetect.commands.quality := TRUE;
   cmCathodeAlignTableElectrodeDetect.monitoring.valid := TRUE;
   cmCathodeAlignTableElectrodeDetect.monitoring.busy := TRUE;
   cmCathodeAlignTableElectrodeDetect.monitoring.error := FALSE;
   cmCathodeAlignTableElectrodeDetect.monitoring.status := 16#0000;
   cmCathodeAlignTableElectrodeDetect.monitoring.risingEdge := FALSE;
   cmCathodeAlignTableElectrodeDetect.monitoring.fallingEdge := FALSE;
   cmCathodeAlignTableElectrodeDetect.monitoring.processValue := FALSE;
   cmCathodeNgPnpElectrodeDetect.commands.reset := FALSE;
   cmCathodeNgPnpElectrodeDetect.commands.simulation := FALSE;
   cmCathodeNgPnpElectrodeDetect.commands.quality := TRUE;
   cmCathodeNgPnpElectrodeDetect.monitoring.valid := FALSE;
   cmCathodeNgPnpElectrodeDetect.monitoring.busy := FALSE;
   cmCathodeNgPnpElectrodeDetect.monitoring.error := FALSE;
   cmCathodeNgPnpElectrodeDetect.monitoring.status := 16#0000;
   cmCathodeNgPnpElectrodeDetect.monitoring.risingEdge := FALSE;
   cmCathodeNgPnpElectrodeDetect.monitoring.fallingEdge := FALSE;
   cmCathodeNgPnpElectrodeDetect.monitoring.processValue := FALSE;
   cmCathodeNgBoxFullSensorDetect.commands.reset := FALSE;
   cmCathodeNgBoxFullSensorDetect.commands.simulation := FALSE;
   cmCathodeNgBoxFullSensorDetect.commands.quality := TRUE;
   cmCathodeNgBoxFullSensorDetect.monitoring.valid := TRUE;
   cmCathodeNgBoxFullSensorDetect.monitoring.busy := TRUE;
   cmCathodeNgBoxFullSensorDetect.monitoring.error := FALSE;
   cmCathodeNgBoxFullSensorDetect.monitoring.status := 16#0000;
   cmCathodeNgBoxFullSensorDetect.monitoring.risingEdge := FALSE;
   cmCathodeNgBoxFullSensorDetect.monitoring.fallingEdge := FALSE;
   cmCathodeNgBoxFullSensorDetect.monitoring.processValue := FALSE;
   cmCathodeNgBoxDetect.commands.reset := FALSE;
   cmCathodeNgBoxDetect.commands.simulation := FALSE;
   cmCathodeNgBoxDetect.commands.quality := TRUE;
   cmCathodeNgBoxDetect.monitoring.valid := TRUE;
   cmCathodeNgBoxDetect.monitoring.busy := TRUE;
   cmCathodeNgBoxDetect.monitoring.error := FALSE;
   cmCathodeNgBoxDetect.monitoring.status := 16#0000;
   cmCathodeNgBoxDetect.monitoring.risingEdge := FALSE;
   cmCathodeNgBoxDetect.monitoring.fallingEdge := FALSE;
   cmCathodeNgBoxDetect.monitoring.processValue := TRUE;
   cmCathodeMainPnP1AxisX.commandConfiguration.generalSettings.stopOnError := TRUE;
   cmCathodeMainPnP1AxisX.commandConfiguration.generalSettings.resetWithRestart := FALSE;
   cmCathodeMainPnP1AxisX.commandConfiguration.generalSettings.abortWaitingSyncCmd := TRUE;
   cmCathodeMainPnP1AxisX.commandConfiguration.power.startMode := 1;
   cmCathodeMainPnP1AxisX.commandConfiguration.power.stopMode := 0;
   cmCathodeMainPnP1AxisX.commandConfiguration.power.syncMotionSimulation := FALSE;
   cmCathodeMainPnP1AxisX.commandConfiguration.power.syncMotionSimulationExtendedMode := -1;
   cmCathodeMainPnP1AxisX.commandConfiguration.jog.velocity := 0.0;
   cmCathodeMainPnP1AxisX.commandConfiguration.jog.acceleration := -1.0;
   cmCathodeMainPnP1AxisX.commandConfiguration.jog.deceleration := -1.0;
   cmCathodeMainPnP1AxisX.commandConfiguration.jog.jerk := -1.0;
   cmCathodeMainPnP1AxisX.commandConfiguration.jog.positionControlled := TRUE;
   cmCathodeMainPnP1AxisX.commandConfiguration.jog.increment := 0.0;
   cmCathodeMainPnP1AxisX.commandConfiguration.jog.mode := 0;
   cmCathodeMainPnP1AxisX.commandConfiguration.moveVelocity.velocity := 0.0;
   cmCathodeMainPnP1AxisX.commandConfiguration.moveVelocity.acceleration := -1.0;
   cmCathodeMainPnP1AxisX.commandConfiguration.moveVelocity.deceleration := -1.0;
   cmCathodeMainPnP1AxisX.commandConfiguration.moveVelocity.jerk := -1.0;
   cmCathodeMainPnP1AxisX.commandConfiguration.moveVelocity.direction := 0;
   cmCathodeMainPnP1AxisX.commandConfiguration.moveVelocity.positionControlled := TRUE;
   cmCathodeMainPnP1AxisX.commandConfiguration.moveVelocity.velocityChangeOnTheFly := FALSE;
   cmCathodeMainPnP1AxisX.commandConfiguration.stop.deceleration := -1.0;
   cmCathodeMainPnP1AxisX.commandConfiguration.stop.jerk := -1.0;
   cmCathodeMainPnP1AxisX.commandConfiguration.stop.abortAcceleration := FALSE;
   cmCathodeMainPnP1AxisX.commandConfiguration.fastStop.deceleration := -1.0;
   cmCathodeMainPnP1AxisX.commandConfiguration.fastStop.jerk := -1.0;
   cmCathodeMainPnP1AxisX.commandConfiguration.fastStop.abortAcceleration := FALSE;
   cmCathodeMainPnP1AxisX.commandConfiguration.fastStop.replaceStopPossible := FALSE;
   cmCathodeMainPnP1AxisX.commandConfiguration.torqueLimiting.limit := -1.0;
   cmCathodeMainPnP1AxisX.commandConfiguration.torqueLimiting.mode := 0;
   cmCathodeMainPnP1AxisX.commandConfiguration.homing.position := 0.0;
   cmCathodeMainPnP1AxisX.commandConfiguration.homing.mode := 0;
   cmCathodeMainPnP1AxisX.commandConfiguration.homing.sensor := 0;
   cmCathodeMainPnP1AxisX.commandConfiguration.homing.extendedMode := -1;
   cmCathodeMainPnP1AxisX.commandConfiguration.homing.extendedModeTorqueLimit := 0.0;
   cmCathodeMainPnP1AxisX.commandConfiguration.homing.extendedModeTargetPosition := 0.0;
   cmCathodeMainPnP1AxisX.commandConfiguration.posRelative.distance := 0.0;
   cmCathodeMainPnP1AxisX.commandConfiguration.posRelative.velocity := -1.0;
   cmCathodeMainPnP1AxisX.commandConfiguration.posRelative.acceleration := -1.0;
   cmCathodeMainPnP1AxisX.commandConfiguration.posRelative.deceleration := -1.0;
   cmCathodeMainPnP1AxisX.commandConfiguration.posRelative.jerk := -1.0;
   cmCathodeMainPnP1AxisX.commandConfiguration.posRelative.direction := 0;
   cmCathodeMainPnP1AxisX.commandConfiguration.posAbsolute.position := 0.0;
   cmCathodeMainPnP1AxisX.commandConfiguration.posAbsolute.velocity := -1.0;
   cmCathodeMainPnP1AxisX.commandConfiguration.posAbsolute.acceleration := -1.0;
   cmCathodeMainPnP1AxisX.commandConfiguration.posAbsolute.deceleration := -1.0;
   cmCathodeMainPnP1AxisX.commandConfiguration.posAbsolute.jerk := -1.0;
   cmCathodeMainPnP1AxisX.commandConfiguration.posAbsolute.direction := 1;
   cmCathodeMainPnP1AxisX.commandConfiguration.posAbsolute.positionChangeOnTheFly := FALSE;
   cmCathodeMainPnP1AxisX.commandConfiguration.posAbsolute.velocityChangeOnTheFly := FALSE;
   cmCathodeMainPnP1AxisX.commandConfiguration.posSuperimposed.distance := 0.0;
   cmCathodeMainPnP1AxisX.commandConfiguration.posSuperimposed.velocityDiff := -1.0;
   cmCathodeMainPnP1AxisX.commandConfiguration.posSuperimposed.acceleration := -1.0;
   cmCathodeMainPnP1AxisX.commandConfiguration.posSuperimposed.deceleration := -1.0;
   cmCathodeMainPnP1AxisX.commandConfiguration.posSuperimposed.jerk := -1.0;
   cmCathodeMainPnP1AxisX.commandConfiguration.posSuperimposed.direction := 0;
   cmCathodeMainPnP1AxisX.commandConfiguration.haltSuperimposed.deceleration := -1.0;
   cmCathodeMainPnP1AxisX.commandConfiguration.haltSuperimposed.jerk := -1.0;
   cmCathodeMainPnP1AxisX.commandConfiguration.haltSuperimposed.abortAcceleration := FALSE;
   cmCathodeMainPnP1AxisX.commandConfiguration.gearInRelative.ratioNumerator := 1;
   cmCathodeMainPnP1AxisX.commandConfiguration.gearInRelative.ratioDenominator := 1;
   cmCathodeMainPnP1AxisX.commandConfiguration.gearInRelative.acceleration := -1.0;
   cmCathodeMainPnP1AxisX.commandConfiguration.gearInRelative.deceleration := -1.0;
   cmCathodeMainPnP1AxisX.commandConfiguration.gearInRelative.jerk := -1.0;
   cmCathodeMainPnP1AxisX.commandConfiguration.gearInRelative.ratioChangeOnTheFly := FALSE;
   cmCathodeMainPnP1AxisX.commandConfiguration.gearInAbsolute.ratioNumerator := 1;
   cmCathodeMainPnP1AxisX.commandConfiguration.gearInAbsolute.ratioDenominator := 1;
   cmCathodeMainPnP1AxisX.commandConfiguration.gearInAbsolute.masterSyncPosition := 0.0;
   cmCathodeMainPnP1AxisX.commandConfiguration.gearInAbsolute.slaveSyncPosition := 0.0;
   cmCathodeMainPnP1AxisX.commandConfiguration.gearInAbsolute.syncProfileReference := 1;
   cmCathodeMainPnP1AxisX.commandConfiguration.gearInAbsolute.masterStartDistance := 0.0;
   cmCathodeMainPnP1AxisX.commandConfiguration.gearInAbsolute.velocity := -1.0;
   cmCathodeMainPnP1AxisX.commandConfiguration.gearInAbsolute.acceleration := -1.0;
   cmCathodeMainPnP1AxisX.commandConfiguration.gearInAbsolute.deceleration := -1.0;
   cmCathodeMainPnP1AxisX.commandConfiguration.gearInAbsolute.jerk := -1.0;
   cmCathodeMainPnP1AxisX.commandConfiguration.gearInAbsolute.syncDirection := 1;
   cmCathodeMainPnP1AxisX.commandConfiguration.gearInAbsolute.ratioChangeOnTheFly := FALSE;
   cmCathodeMainPnP1AxisX.commandConfiguration.gearInVelocity.continuousUpdate := FALSE;
   cmCathodeMainPnP1AxisX.commandConfiguration.gearInVelocity.ratioNumerator := 1;
   cmCathodeMainPnP1AxisX.commandConfiguration.gearInVelocity.ratioDenominator := 1;
   cmCathodeMainPnP1AxisX.commandConfiguration.gearInVelocity.acceleration := -1.0;
   cmCathodeMainPnP1AxisX.commandConfiguration.gearInVelocity.deceleration := -1.0;
   cmCathodeMainPnP1AxisX.commandConfiguration.gearInVelocity.jerk := -1.0;
   cmCathodeMainPnP1AxisX.commandConfiguration.gearInVelocity.positionControlled := FALSE;
   cmCathodeMainPnP1AxisX.commandConfiguration.camIn.masterOffset := 0.0;
   cmCathodeMainPnP1AxisX.commandConfiguration.camIn.slaveOffset := 0.0;
   cmCathodeMainPnP1AxisX.commandConfiguration.camIn.masterScaling := 1.0;
   cmCathodeMainPnP1AxisX.commandConfiguration.camIn.slaveScaling := 1.0;
   cmCathodeMainPnP1AxisX.commandConfiguration.camIn.masterSyncPosition := 0.0;
   cmCathodeMainPnP1AxisX.commandConfiguration.camIn.syncProfileReference := 1;
   cmCathodeMainPnP1AxisX.commandConfiguration.camIn.masterStartDistance := 0.0;
   cmCathodeMainPnP1AxisX.commandConfiguration.camIn.velocity := -1.0;
   cmCathodeMainPnP1AxisX.commandConfiguration.camIn.acceleration := -1.0;
   cmCathodeMainPnP1AxisX.commandConfiguration.camIn.deceleration := -1.0;
   cmCathodeMainPnP1AxisX.commandConfiguration.camIn.jerk := -1.0;
   cmCathodeMainPnP1AxisX.commandConfiguration.camIn.applicationMode := 0;
   cmCathodeMainPnP1AxisX.commandConfiguration.camIn.syncDirection := 1;
   cmCathodeMainPnP1AxisX.commandConfiguration.gearOutCamOut.slavePosition := 0.0;
   cmCathodeMainPnP1AxisX.commandConfiguration.gearOutCamOut.syncProfileReference := 1;
   cmCathodeMainPnP1AxisX.commandConfiguration.gearOutCamOut.masterStopDistance := 0.0;
   cmCathodeMainPnP1AxisX.commandConfiguration.gearOutCamOut.deceleration := -1.0;
   cmCathodeMainPnP1AxisX.commandConfiguration.gearOutCamOut.jerk := -1.0;
   cmCathodeMainPnP1AxisX.commandConfiguration.gearOutCamOut.syncOutDirection := 3;
   cmCathodeMainPnP1AxisX.commandConfiguration.gearOutCamOut.gearOutCamOutMode := -1;
   cmCathodeMainPnP1AxisX.commandConfiguration.phasing.phaseShift := 0.0;
   cmCathodeMainPnP1AxisX.commandConfiguration.phasing.velocity := -1.0;
   cmCathodeMainPnP1AxisX.commandConfiguration.phasing.acceleration := -1.0;
   cmCathodeMainPnP1AxisX.commandConfiguration.phasing.deceleration := -1.0;
   cmCathodeMainPnP1AxisX.commandConfiguration.phasing.jerk := -1.0;
   cmCathodeMainPnP1AxisX.commandConfiguration.phasing.profileReference := 0;
   cmCathodeMainPnP1AxisX.commandConfiguration.phasing.phasingDistance := 0.0;
   cmCathodeMainPnP1AxisX.commandConfiguration.phasing.startPosition := 0.0;
   cmCathodeMainPnP1AxisX.commandConfiguration.phasing.direction := 3;
   cmCathodeMainPnP1AxisX.commandConfiguration.phasing.phaseAbsolute := TRUE;
   cmCathodeMainPnP1AxisX.commandConfiguration.phasing.phaseShiftChangeOnTheFly := FALSE;
   cmCathodeMainPnP1AxisX.commandConfiguration.offset.offset := 0.0;
   cmCathodeMainPnP1AxisX.commandConfiguration.offset.profileReference := 1;
   cmCathodeMainPnP1AxisX.commandConfiguration.offset.offsetDistance := 0.0;
   cmCathodeMainPnP1AxisX.commandConfiguration.offset.startPosition := 0.0;
   cmCathodeMainPnP1AxisX.commandConfiguration.offset.direction := 3;
   cmCathodeMainPnP1AxisX.commandConfiguration.offset.offsetAbsolute := TRUE;
   cmCathodeMainPnP1AxisX.commandConfiguration.offset.offsetChangeOnTheFly := FALSE;
   cmCathodeMainPnP1AxisX.commands.enableAxis := FALSE;
   cmCathodeMainPnP1AxisX.commands.resetAxis := FALSE;
   cmCathodeMainPnP1AxisX.commands.openBrake := FALSE;
   cmCathodeMainPnP1AxisX.commands.jogForward := FALSE;
   cmCathodeMainPnP1AxisX.commands.jogBackward := FALSE;
   cmCathodeMainPnP1AxisX.commands.moveVelocity := FALSE;
   cmCathodeMainPnP1AxisX.commands.stop := FALSE;
   cmCathodeMainPnP1AxisX.commands.fastStop := FALSE;
   cmCathodeMainPnP1AxisX.commands.torqueLimiting := FALSE;
   cmCathodeMainPnP1AxisX.commands.homing := FALSE;
   cmCathodeMainPnP1AxisX.commands.posRelative := FALSE;
   cmCathodeMainPnP1AxisX.commands.posAbsolute := FALSE;
   cmCathodeMainPnP1AxisX.commands.posSuperimposed := FALSE;
   cmCathodeMainPnP1AxisX.commands.haltSuperimposed := FALSE;
   cmCathodeMainPnP1AxisX.commands.selectSetPosition := -1;
   cmCathodeMainPnP1AxisX.commands.reset := FALSE;
   cmCathodeMainPnP1AxisX.monitoring.valid := FALSE;
   cmCathodeMainPnP1AxisX.monitoring.busy := TRUE;
   cmCathodeMainPnP1AxisX.monitoring.error := TRUE;
   cmCathodeMainPnP1AxisX.monitoring.status := 16#8600;
   cmCathodeMainPnP1AxisX.monitoring.subfunctionStatus := 16#8001;
   cmCathodeMainPnP1AxisX.monitoring.axisEnabled := FALSE;
   cmCathodeMainPnP1AxisX.monitoring.resetActive := FALSE;
   cmCathodeMainPnP1AxisX.monitoring.inVelocity := FALSE;
   cmCathodeMainPnP1AxisX.monitoring.inLimitation := FALSE;
   cmCathodeMainPnP1AxisX.monitoring.inClamping := FALSE;
   cmCathodeMainPnP1AxisX.monitoring.startSync := FALSE;
   cmCathodeMainPnP1AxisX.monitoring.inSync := FALSE;
   cmCathodeMainPnP1AxisX.monitoring.inSimulation := FALSE;
   cmCathodeMainPnP1AxisX.monitoring.jogSelected := FALSE;
   cmCathodeMainPnP1AxisX.monitoring.moveVelocitySelected := FALSE;
   cmCathodeMainPnP1AxisX.monitoring.stopSelected := FALSE;
   cmCathodeMainPnP1AxisX.monitoring.fastStopSelected := FALSE;
   cmCathodeMainPnP1AxisX.monitoring.torqueLimitingSelected := FALSE;
   cmCathodeMainPnP1AxisX.monitoring.homingSelected := FALSE;
   cmCathodeMainPnP1AxisX.monitoring.posRelativeSelected := FALSE;
   cmCathodeMainPnP1AxisX.monitoring.posAbsoluteSelected := FALSE;
   cmCathodeMainPnP1AxisX.monitoring.posSuperimposedSelected := FALSE;
   cmCathodeMainPnP1AxisX.monitoring.haltSuperimposedSelected := FALSE;
   cmCathodeMainPnP1AxisX.monitoring.commandBusy := FALSE;
   cmCathodeMainPnP1AxisX.monitoring.commandDone := FALSE;
   cmCathodeMainPnP1AxisX.monitoring.commandAborted := FALSE;
   cmCathodeMainPnP1AxisX.monitoring.homingCommandBusy := FALSE;
   cmCathodeMainPnP1AxisX.monitoring.homingCommandDone := FALSE;
   cmCathodeMainPnP1AxisX.monitoring.homingCommandAborted := FALSE;
   cmCathodeMainPnP1AxisX.monitoring.superimposedBusy := FALSE;
   cmCathodeMainPnP1AxisX.monitoring.superimposedDone := FALSE;
   cmCathodeMainPnP1AxisX.monitoring.superimposedAborted := FALSE;
   cmCathodeMainPnP1AxisX.monitoring.actualPosition := 0.048;
   cmCathodeMainPnP1AxisX.monitoring.actualSpeed := 0.0;
   cmCathodeMainPnP1AxisX.monitoring.speedUnit := 1062;
   cmCathodeMainPnP1AxisX.monitoring.positionUnit := 1013;
   cmCathodeMainPnP1AxisX.monitoring.axisType := 1;
   cmCathodeMainPnP1AxisX.monitoring.interlockGeneralOut := TRUE;
   cmCathodeMainPnP1AxisX.monitoring.interlockJogForwardOut := TRUE;
   cmCathodeMainPnP1AxisX.monitoring.interlockJogBackwardOut := TRUE;
   cmCathodeMainPnP2AxisX.commandConfiguration.generalSettings.stopOnError := TRUE;
   cmCathodeMainPnP2AxisX.commandConfiguration.generalSettings.resetWithRestart := FALSE;
   cmCathodeMainPnP2AxisX.commandConfiguration.generalSettings.abortWaitingSyncCmd := TRUE;
   cmCathodeMainPnP2AxisX.commandConfiguration.power.startMode := 1;
   cmCathodeMainPnP2AxisX.commandConfiguration.power.stopMode := 0;
   cmCathodeMainPnP2AxisX.commandConfiguration.power.syncMotionSimulation := FALSE;
   cmCathodeMainPnP2AxisX.commandConfiguration.power.syncMotionSimulationExtendedMode := -1;
   cmCathodeMainPnP2AxisX.commandConfiguration.jog.velocity := 0.0;
   cmCathodeMainPnP2AxisX.commandConfiguration.jog.acceleration := -1.0;
   cmCathodeMainPnP2AxisX.commandConfiguration.jog.deceleration := -1.0;
   cmCathodeMainPnP2AxisX.commandConfiguration.jog.jerk := -1.0;
   cmCathodeMainPnP2AxisX.commandConfiguration.jog.positionControlled := TRUE;
   cmCathodeMainPnP2AxisX.commandConfiguration.jog.increment := 0.0;
   cmCathodeMainPnP2AxisX.commandConfiguration.jog.mode := 0;
   cmCathodeMainPnP2AxisX.commandConfiguration.moveVelocity.velocity := 0.0;
   cmCathodeMainPnP2AxisX.commandConfiguration.moveVelocity.acceleration := -1.0;
   cmCathodeMainPnP2AxisX.commandConfiguration.moveVelocity.deceleration := -1.0;
   cmCathodeMainPnP2AxisX.commandConfiguration.moveVelocity.jerk := -1.0;
   cmCathodeMainPnP2AxisX.commandConfiguration.moveVelocity.direction := 0;
   cmCathodeMainPnP2AxisX.commandConfiguration.moveVelocity.positionControlled := TRUE;
   cmCathodeMainPnP2AxisX.commandConfiguration.moveVelocity.velocityChangeOnTheFly := FALSE;
   cmCathodeMainPnP2AxisX.commandConfiguration.stop.deceleration := -1.0;
   cmCathodeMainPnP2AxisX.commandConfiguration.stop.jerk := -1.0;
   cmCathodeMainPnP2AxisX.commandConfiguration.stop.abortAcceleration := FALSE;
   cmCathodeMainPnP2AxisX.commandConfiguration.fastStop.deceleration := -1.0;
   cmCathodeMainPnP2AxisX.commandConfiguration.fastStop.jerk := -1.0;
   cmCathodeMainPnP2AxisX.commandConfiguration.fastStop.abortAcceleration := FALSE;
   cmCathodeMainPnP2AxisX.commandConfiguration.fastStop.replaceStopPossible := FALSE;
   cmCathodeMainPnP2AxisX.commandConfiguration.torqueLimiting.limit := -1.0;
   cmCathodeMainPnP2AxisX.commandConfiguration.torqueLimiting.mode := 0;
   cmCathodeMainPnP2AxisX.commandConfiguration.homing.position := 0.0;
   cmCathodeMainPnP2AxisX.commandConfiguration.homing.mode := 0;
   cmCathodeMainPnP2AxisX.commandConfiguration.homing.sensor := 0;
   cmCathodeMainPnP2AxisX.commandConfiguration.homing.extendedMode := -1;
   cmCathodeMainPnP2AxisX.commandConfiguration.homing.extendedModeTorqueLimit := 0.0;
   cmCathodeMainPnP2AxisX.commandConfiguration.homing.extendedModeTargetPosition := 0.0;
   cmCathodeMainPnP2AxisX.commandConfiguration.posRelative.distance := 0.0;
   cmCathodeMainPnP2AxisX.commandConfiguration.posRelative.velocity := -1.0;
   cmCathodeMainPnP2AxisX.commandConfiguration.posRelative.acceleration := -1.0;
   cmCathodeMainPnP2AxisX.commandConfiguration.posRelative.deceleration := -1.0;
   cmCathodeMainPnP2AxisX.commandConfiguration.posRelative.jerk := -1.0;
   cmCathodeMainPnP2AxisX.commandConfiguration.posRelative.direction := 0;
   cmCathodeMainPnP2AxisX.commandConfiguration.posAbsolute.position := 0.0;
   cmCathodeMainPnP2AxisX.commandConfiguration.posAbsolute.velocity := -1.0;
   cmCathodeMainPnP2AxisX.commandConfiguration.posAbsolute.acceleration := -1.0;
   cmCathodeMainPnP2AxisX.commandConfiguration.posAbsolute.deceleration := -1.0;
   cmCathodeMainPnP2AxisX.commandConfiguration.posAbsolute.jerk := -1.0;
   cmCathodeMainPnP2AxisX.commandConfiguration.posAbsolute.direction := 1;
   cmCathodeMainPnP2AxisX.commandConfiguration.posAbsolute.positionChangeOnTheFly := FALSE;
   cmCathodeMainPnP2AxisX.commandConfiguration.posAbsolute.velocityChangeOnTheFly := FALSE;
   cmCathodeMainPnP2AxisX.commandConfiguration.posSuperimposed.distance := 0.0;
   cmCathodeMainPnP2AxisX.commandConfiguration.posSuperimposed.velocityDiff := -1.0;
   cmCathodeMainPnP2AxisX.commandConfiguration.posSuperimposed.acceleration := -1.0;
   cmCathodeMainPnP2AxisX.commandConfiguration.posSuperimposed.deceleration := -1.0;
   cmCathodeMainPnP2AxisX.commandConfiguration.posSuperimposed.jerk := -1.0;
   cmCathodeMainPnP2AxisX.commandConfiguration.posSuperimposed.direction := 0;
   cmCathodeMainPnP2AxisX.commandConfiguration.haltSuperimposed.deceleration := -1.0;
   cmCathodeMainPnP2AxisX.commandConfiguration.haltSuperimposed.jerk := -1.0;
   cmCathodeMainPnP2AxisX.commandConfiguration.haltSuperimposed.abortAcceleration := FALSE;
   cmCathodeMainPnP2AxisX.commandConfiguration.gearInRelative.ratioNumerator := 1;
   cmCathodeMainPnP2AxisX.commandConfiguration.gearInRelative.ratioDenominator := 1;
   cmCathodeMainPnP2AxisX.commandConfiguration.gearInRelative.acceleration := -1.0;
   cmCathodeMainPnP2AxisX.commandConfiguration.gearInRelative.deceleration := -1.0;
   cmCathodeMainPnP2AxisX.commandConfiguration.gearInRelative.jerk := -1.0;
   cmCathodeMainPnP2AxisX.commandConfiguration.gearInRelative.ratioChangeOnTheFly := FALSE;
   cmCathodeMainPnP2AxisX.commandConfiguration.gearInAbsolute.ratioNumerator := 1;
   cmCathodeMainPnP2AxisX.commandConfiguration.gearInAbsolute.ratioDenominator := 1;
   cmCathodeMainPnP2AxisX.commandConfiguration.gearInAbsolute.masterSyncPosition := 0.0;
   cmCathodeMainPnP2AxisX.commandConfiguration.gearInAbsolute.slaveSyncPosition := 0.0;
   cmCathodeMainPnP2AxisX.commandConfiguration.gearInAbsolute.syncProfileReference := 1;
   cmCathodeMainPnP2AxisX.commandConfiguration.gearInAbsolute.masterStartDistance := 0.0;
   cmCathodeMainPnP2AxisX.commandConfiguration.gearInAbsolute.velocity := -1.0;
   cmCathodeMainPnP2AxisX.commandConfiguration.gearInAbsolute.acceleration := -1.0;
   cmCathodeMainPnP2AxisX.commandConfiguration.gearInAbsolute.deceleration := -1.0;
   cmCathodeMainPnP2AxisX.commandConfiguration.gearInAbsolute.jerk := -1.0;
   cmCathodeMainPnP2AxisX.commandConfiguration.gearInAbsolute.syncDirection := 1;
   cmCathodeMainPnP2AxisX.commandConfiguration.gearInAbsolute.ratioChangeOnTheFly := FALSE;
   cmCathodeMainPnP2AxisX.commandConfiguration.gearInVelocity.continuousUpdate := FALSE;
   cmCathodeMainPnP2AxisX.commandConfiguration.gearInVelocity.ratioNumerator := 1;
   cmCathodeMainPnP2AxisX.commandConfiguration.gearInVelocity.ratioDenominator := 1;
   cmCathodeMainPnP2AxisX.commandConfiguration.gearInVelocity.acceleration := -1.0;
   cmCathodeMainPnP2AxisX.commandConfiguration.gearInVelocity.deceleration := -1.0;
   cmCathodeMainPnP2AxisX.commandConfiguration.gearInVelocity.jerk := -1.0;
   cmCathodeMainPnP2AxisX.commandConfiguration.gearInVelocity.positionControlled := FALSE;
   cmCathodeMainPnP2AxisX.commandConfiguration.camIn.masterOffset := 0.0;
   cmCathodeMainPnP2AxisX.commandConfiguration.camIn.slaveOffset := 0.0;
   cmCathodeMainPnP2AxisX.commandConfiguration.camIn.masterScaling := 1.0;
   cmCathodeMainPnP2AxisX.commandConfiguration.camIn.slaveScaling := 1.0;
   cmCathodeMainPnP2AxisX.commandConfiguration.camIn.masterSyncPosition := 0.0;
   cmCathodeMainPnP2AxisX.commandConfiguration.camIn.syncProfileReference := 1;
   cmCathodeMainPnP2AxisX.commandConfiguration.camIn.masterStartDistance := 0.0;
   cmCathodeMainPnP2AxisX.commandConfiguration.camIn.velocity := -1.0;
   cmCathodeMainPnP2AxisX.commandConfiguration.camIn.acceleration := -1.0;
   cmCathodeMainPnP2AxisX.commandConfiguration.camIn.deceleration := -1.0;
   cmCathodeMainPnP2AxisX.commandConfiguration.camIn.jerk := -1.0;
   cmCathodeMainPnP2AxisX.commandConfiguration.camIn.applicationMode := 0;
   cmCathodeMainPnP2AxisX.commandConfiguration.camIn.syncDirection := 1;
   cmCathodeMainPnP2AxisX.commandConfiguration.gearOutCamOut.slavePosition := 0.0;
   cmCathodeMainPnP2AxisX.commandConfiguration.gearOutCamOut.syncProfileReference := 1;
   cmCathodeMainPnP2AxisX.commandConfiguration.gearOutCamOut.masterStopDistance := 0.0;
   cmCathodeMainPnP2AxisX.commandConfiguration.gearOutCamOut.deceleration := -1.0;
   cmCathodeMainPnP2AxisX.commandConfiguration.gearOutCamOut.jerk := -1.0;
   cmCathodeMainPnP2AxisX.commandConfiguration.gearOutCamOut.syncOutDirection := 3;
   cmCathodeMainPnP2AxisX.commandConfiguration.gearOutCamOut.gearOutCamOutMode := -1;
   cmCathodeMainPnP2AxisX.commandConfiguration.phasing.phaseShift := 0.0;
   cmCathodeMainPnP2AxisX.commandConfiguration.phasing.velocity := -1.0;
   cmCathodeMainPnP2AxisX.commandConfiguration.phasing.acceleration := -1.0;
   cmCathodeMainPnP2AxisX.commandConfiguration.phasing.deceleration := -1.0;
   cmCathodeMainPnP2AxisX.commandConfiguration.phasing.jerk := -1.0;
   cmCathodeMainPnP2AxisX.commandConfiguration.phasing.profileReference := 0;
   cmCathodeMainPnP2AxisX.commandConfiguration.phasing.phasingDistance := 0.0;
   cmCathodeMainPnP2AxisX.commandConfiguration.phasing.startPosition := 0.0;
   cmCathodeMainPnP2AxisX.commandConfiguration.phasing.direction := 3;
   cmCathodeMainPnP2AxisX.commandConfiguration.phasing.phaseAbsolute := TRUE;
   cmCathodeMainPnP2AxisX.commandConfiguration.phasing.phaseShiftChangeOnTheFly := FALSE;
   cmCathodeMainPnP2AxisX.commandConfiguration.offset.offset := 0.0;
   cmCathodeMainPnP2AxisX.commandConfiguration.offset.profileReference := 1;
   cmCathodeMainPnP2AxisX.commandConfiguration.offset.offsetDistance := 0.0;
   cmCathodeMainPnP2AxisX.commandConfiguration.offset.startPosition := 0.0;
   cmCathodeMainPnP2AxisX.commandConfiguration.offset.direction := 3;
   cmCathodeMainPnP2AxisX.commandConfiguration.offset.offsetAbsolute := TRUE;
   cmCathodeMainPnP2AxisX.commandConfiguration.offset.offsetChangeOnTheFly := FALSE;
   cmCathodeMainPnP2AxisX.commands.enableAxis := FALSE;
   cmCathodeMainPnP2AxisX.commands.resetAxis := FALSE;
   cmCathodeMainPnP2AxisX.commands.openBrake := FALSE;
   cmCathodeMainPnP2AxisX.commands.jogForward := FALSE;
   cmCathodeMainPnP2AxisX.commands.jogBackward := FALSE;
   cmCathodeMainPnP2AxisX.commands.moveVelocity := FALSE;
   cmCathodeMainPnP2AxisX.commands.stop := FALSE;
   cmCathodeMainPnP2AxisX.commands.fastStop := FALSE;
   cmCathodeMainPnP2AxisX.commands.torqueLimiting := FALSE;
   cmCathodeMainPnP2AxisX.commands.homing := FALSE;
   cmCathodeMainPnP2AxisX.commands.posRelative := FALSE;
   cmCathodeMainPnP2AxisX.commands.posAbsolute := FALSE;
   cmCathodeMainPnP2AxisX.commands.posSuperimposed := FALSE;
   cmCathodeMainPnP2AxisX.commands.haltSuperimposed := FALSE;
   cmCathodeMainPnP2AxisX.commands.selectSetPosition := -1;
   cmCathodeMainPnP2AxisX.commands.reset := FALSE;
   cmCathodeMainPnP2AxisX.monitoring.valid := FALSE;
   cmCathodeMainPnP2AxisX.monitoring.busy := TRUE;
   cmCathodeMainPnP2AxisX.monitoring.error := TRUE;
   cmCathodeMainPnP2AxisX.monitoring.status := 16#8600;
   cmCathodeMainPnP2AxisX.monitoring.subfunctionStatus := 16#8001;
   cmCathodeMainPnP2AxisX.monitoring.axisEnabled := FALSE;
   cmCathodeMainPnP2AxisX.monitoring.resetActive := FALSE;
   cmCathodeMainPnP2AxisX.monitoring.inVelocity := FALSE;
   cmCathodeMainPnP2AxisX.monitoring.inLimitation := FALSE;
   cmCathodeMainPnP2AxisX.monitoring.inClamping := FALSE;
   cmCathodeMainPnP2AxisX.monitoring.startSync := FALSE;
   cmCathodeMainPnP2AxisX.monitoring.inSync := FALSE;
   cmCathodeMainPnP2AxisX.monitoring.inSimulation := FALSE;
   cmCathodeMainPnP2AxisX.monitoring.jogSelected := FALSE;
   cmCathodeMainPnP2AxisX.monitoring.moveVelocitySelected := FALSE;
   cmCathodeMainPnP2AxisX.monitoring.stopSelected := FALSE;
   cmCathodeMainPnP2AxisX.monitoring.fastStopSelected := FALSE;
   cmCathodeMainPnP2AxisX.monitoring.torqueLimitingSelected := FALSE;
   cmCathodeMainPnP2AxisX.monitoring.homingSelected := FALSE;
   cmCathodeMainPnP2AxisX.monitoring.posRelativeSelected := FALSE;
   cmCathodeMainPnP2AxisX.monitoring.posAbsoluteSelected := FALSE;
   cmCathodeMainPnP2AxisX.monitoring.posSuperimposedSelected := FALSE;
   cmCathodeMainPnP2AxisX.monitoring.haltSuperimposedSelected := FALSE;
   cmCathodeMainPnP2AxisX.monitoring.commandBusy := FALSE;
   cmCathodeMainPnP2AxisX.monitoring.commandDone := FALSE;
   cmCathodeMainPnP2AxisX.monitoring.commandAborted := FALSE;
   cmCathodeMainPnP2AxisX.monitoring.homingCommandBusy := FALSE;
   cmCathodeMainPnP2AxisX.monitoring.homingCommandDone := FALSE;
   cmCathodeMainPnP2AxisX.monitoring.homingCommandAborted := FALSE;
   cmCathodeMainPnP2AxisX.monitoring.superimposedBusy := FALSE;
   cmCathodeMainPnP2AxisX.monitoring.superimposedDone := FALSE;
   cmCathodeMainPnP2AxisX.monitoring.superimposedAborted := FALSE;
   cmCathodeMainPnP2AxisX.monitoring.actualPosition := -11.988;
   cmCathodeMainPnP2AxisX.monitoring.actualSpeed := -0.000333333333333333;
   cmCathodeMainPnP2AxisX.monitoring.speedUnit := 1062;
   cmCathodeMainPnP2AxisX.monitoring.positionUnit := 1013;
   cmCathodeMainPnP2AxisX.monitoring.axisType := 1;
   cmCathodeMainPnP2AxisX.monitoring.interlockGeneralOut := TRUE;
   cmCathodeMainPnP2AxisX.monitoring.interlockJogForwardOut := TRUE;
   cmCathodeMainPnP2AxisX.monitoring.interlockJogBackwardOut := TRUE;
   cmCathodeMainPnP1AxisY.commandConfiguration.generalSettings.stopOnError := TRUE;
   cmCathodeMainPnP1AxisY.commandConfiguration.generalSettings.resetWithRestart := FALSE;
   cmCathodeMainPnP1AxisY.commandConfiguration.generalSettings.abortWaitingSyncCmd := TRUE;
   cmCathodeMainPnP1AxisY.commandConfiguration.power.startMode := 1;
   cmCathodeMainPnP1AxisY.commandConfiguration.power.stopMode := 0;
   cmCathodeMainPnP1AxisY.commandConfiguration.power.syncMotionSimulation := FALSE;
   cmCathodeMainPnP1AxisY.commandConfiguration.power.syncMotionSimulationExtendedMode := -1;
   cmCathodeMainPnP1AxisY.commandConfiguration.jog.velocity := 0.0;
   cmCathodeMainPnP1AxisY.commandConfiguration.jog.acceleration := -1.0;
   cmCathodeMainPnP1AxisY.commandConfiguration.jog.deceleration := -1.0;
   cmCathodeMainPnP1AxisY.commandConfiguration.jog.jerk := -1.0;
   cmCathodeMainPnP1AxisY.commandConfiguration.jog.positionControlled := TRUE;
   cmCathodeMainPnP1AxisY.commandConfiguration.jog.increment := 0.0;
   cmCathodeMainPnP1AxisY.commandConfiguration.jog.mode := 0;
   cmCathodeMainPnP1AxisY.commandConfiguration.moveVelocity.velocity := 0.0;
   cmCathodeMainPnP1AxisY.commandConfiguration.moveVelocity.acceleration := -1.0;
   cmCathodeMainPnP1AxisY.commandConfiguration.moveVelocity.deceleration := -1.0;
   cmCathodeMainPnP1AxisY.commandConfiguration.moveVelocity.jerk := -1.0;
   cmCathodeMainPnP1AxisY.commandConfiguration.moveVelocity.direction := 0;
   cmCathodeMainPnP1AxisY.commandConfiguration.moveVelocity.positionControlled := TRUE;
   cmCathodeMainPnP1AxisY.commandConfiguration.moveVelocity.velocityChangeOnTheFly := FALSE;
   cmCathodeMainPnP1AxisY.commandConfiguration.stop.deceleration := -1.0;
   cmCathodeMainPnP1AxisY.commandConfiguration.stop.jerk := -1.0;
   cmCathodeMainPnP1AxisY.commandConfiguration.stop.abortAcceleration := FALSE;
   cmCathodeMainPnP1AxisY.commandConfiguration.fastStop.deceleration := -1.0;
   cmCathodeMainPnP1AxisY.commandConfiguration.fastStop.jerk := -1.0;
   cmCathodeMainPnP1AxisY.commandConfiguration.fastStop.abortAcceleration := FALSE;
   cmCathodeMainPnP1AxisY.commandConfiguration.fastStop.replaceStopPossible := FALSE;
   cmCathodeMainPnP1AxisY.commandConfiguration.torqueLimiting.limit := -1.0;
   cmCathodeMainPnP1AxisY.commandConfiguration.torqueLimiting.mode := 0;
   cmCathodeMainPnP1AxisY.commandConfiguration.homing.position := 0.0;
   cmCathodeMainPnP1AxisY.commandConfiguration.homing.mode := 0;
   cmCathodeMainPnP1AxisY.commandConfiguration.homing.sensor := 0;
   cmCathodeMainPnP1AxisY.commandConfiguration.homing.extendedMode := -1;
   cmCathodeMainPnP1AxisY.commandConfiguration.homing.extendedModeTorqueLimit := 0.0;
   cmCathodeMainPnP1AxisY.commandConfiguration.homing.extendedModeTargetPosition := 0.0;
   cmCathodeMainPnP1AxisY.commandConfiguration.posRelative.distance := 0.0;
   cmCathodeMainPnP1AxisY.commandConfiguration.posRelative.velocity := -1.0;
   cmCathodeMainPnP1AxisY.commandConfiguration.posRelative.acceleration := -1.0;
   cmCathodeMainPnP1AxisY.commandConfiguration.posRelative.deceleration := -1.0;
   cmCathodeMainPnP1AxisY.commandConfiguration.posRelative.jerk := -1.0;
   cmCathodeMainPnP1AxisY.commandConfiguration.posRelative.direction := 0;
   cmCathodeMainPnP1AxisY.commandConfiguration.posAbsolute.position := 0.0;
   cmCathodeMainPnP1AxisY.commandConfiguration.posAbsolute.velocity := -1.0;
   cmCathodeMainPnP1AxisY.commandConfiguration.posAbsolute.acceleration := -1.0;
   cmCathodeMainPnP1AxisY.commandConfiguration.posAbsolute.deceleration := -1.0;
   cmCathodeMainPnP1AxisY.commandConfiguration.posAbsolute.jerk := -1.0;
   cmCathodeMainPnP1AxisY.commandConfiguration.posAbsolute.direction := 1;
   cmCathodeMainPnP1AxisY.commandConfiguration.posAbsolute.positionChangeOnTheFly := FALSE;
   cmCathodeMainPnP1AxisY.commandConfiguration.posAbsolute.velocityChangeOnTheFly := FALSE;
   cmCathodeMainPnP1AxisY.commandConfiguration.posSuperimposed.distance := 0.0;
   cmCathodeMainPnP1AxisY.commandConfiguration.posSuperimposed.velocityDiff := -1.0;
   cmCathodeMainPnP1AxisY.commandConfiguration.posSuperimposed.acceleration := -1.0;
   cmCathodeMainPnP1AxisY.commandConfiguration.posSuperimposed.deceleration := -1.0;
   cmCathodeMainPnP1AxisY.commandConfiguration.posSuperimposed.jerk := -1.0;
   cmCathodeMainPnP1AxisY.commandConfiguration.posSuperimposed.direction := 0;
   cmCathodeMainPnP1AxisY.commandConfiguration.haltSuperimposed.deceleration := -1.0;
   cmCathodeMainPnP1AxisY.commandConfiguration.haltSuperimposed.jerk := -1.0;
   cmCathodeMainPnP1AxisY.commandConfiguration.haltSuperimposed.abortAcceleration := FALSE;
   cmCathodeMainPnP1AxisY.commandConfiguration.gearInRelative.ratioNumerator := 1;
   cmCathodeMainPnP1AxisY.commandConfiguration.gearInRelative.ratioDenominator := 1;
   cmCathodeMainPnP1AxisY.commandConfiguration.gearInRelative.acceleration := -1.0;
   cmCathodeMainPnP1AxisY.commandConfiguration.gearInRelative.deceleration := -1.0;
   cmCathodeMainPnP1AxisY.commandConfiguration.gearInRelative.jerk := -1.0;
   cmCathodeMainPnP1AxisY.commandConfiguration.gearInRelative.ratioChangeOnTheFly := FALSE;
   cmCathodeMainPnP1AxisY.commandConfiguration.gearInAbsolute.ratioNumerator := 1;
   cmCathodeMainPnP1AxisY.commandConfiguration.gearInAbsolute.ratioDenominator := 1;
   cmCathodeMainPnP1AxisY.commandConfiguration.gearInAbsolute.masterSyncPosition := 0.0;
   cmCathodeMainPnP1AxisY.commandConfiguration.gearInAbsolute.slaveSyncPosition := 0.0;
   cmCathodeMainPnP1AxisY.commandConfiguration.gearInAbsolute.syncProfileReference := 1;
   cmCathodeMainPnP1AxisY.commandConfiguration.gearInAbsolute.masterStartDistance := 0.0;
   cmCathodeMainPnP1AxisY.commandConfiguration.gearInAbsolute.velocity := -1.0;
   cmCathodeMainPnP1AxisY.commandConfiguration.gearInAbsolute.acceleration := -1.0;
   cmCathodeMainPnP1AxisY.commandConfiguration.gearInAbsolute.deceleration := -1.0;
   cmCathodeMainPnP1AxisY.commandConfiguration.gearInAbsolute.jerk := -1.0;
   cmCathodeMainPnP1AxisY.commandConfiguration.gearInAbsolute.syncDirection := 1;
   cmCathodeMainPnP1AxisY.commandConfiguration.gearInAbsolute.ratioChangeOnTheFly := FALSE;
   cmCathodeMainPnP1AxisY.commandConfiguration.gearInVelocity.continuousUpdate := FALSE;
   cmCathodeMainPnP1AxisY.commandConfiguration.gearInVelocity.ratioNumerator := 1;
   cmCathodeMainPnP1AxisY.commandConfiguration.gearInVelocity.ratioDenominator := 1;
   cmCathodeMainPnP1AxisY.commandConfiguration.gearInVelocity.acceleration := -1.0;
   cmCathodeMainPnP1AxisY.commandConfiguration.gearInVelocity.deceleration := -1.0;
   cmCathodeMainPnP1AxisY.commandConfiguration.gearInVelocity.jerk := -1.0;
   cmCathodeMainPnP1AxisY.commandConfiguration.gearInVelocity.positionControlled := FALSE;
   cmCathodeMainPnP1AxisY.commandConfiguration.camIn.masterOffset := 0.0;
   cmCathodeMainPnP1AxisY.commandConfiguration.camIn.slaveOffset := 0.0;
   cmCathodeMainPnP1AxisY.commandConfiguration.camIn.masterScaling := 1.0;
   cmCathodeMainPnP1AxisY.commandConfiguration.camIn.slaveScaling := 1.0;
   cmCathodeMainPnP1AxisY.commandConfiguration.camIn.masterSyncPosition := 0.0;
   cmCathodeMainPnP1AxisY.commandConfiguration.camIn.syncProfileReference := 1;
   cmCathodeMainPnP1AxisY.commandConfiguration.camIn.masterStartDistance := 0.0;
   cmCathodeMainPnP1AxisY.commandConfiguration.camIn.velocity := -1.0;
   cmCathodeMainPnP1AxisY.commandConfiguration.camIn.acceleration := -1.0;
   cmCathodeMainPnP1AxisY.commandConfiguration.camIn.deceleration := -1.0;
   cmCathodeMainPnP1AxisY.commandConfiguration.camIn.jerk := -1.0;
   cmCathodeMainPnP1AxisY.commandConfiguration.camIn.applicationMode := 0;
   cmCathodeMainPnP1AxisY.commandConfiguration.camIn.syncDirection := 1;
   cmCathodeMainPnP1AxisY.commandConfiguration.gearOutCamOut.slavePosition := 0.0;
   cmCathodeMainPnP1AxisY.commandConfiguration.gearOutCamOut.syncProfileReference := 1;
   cmCathodeMainPnP1AxisY.commandConfiguration.gearOutCamOut.masterStopDistance := 0.0;
   cmCathodeMainPnP1AxisY.commandConfiguration.gearOutCamOut.deceleration := -1.0;
   cmCathodeMainPnP1AxisY.commandConfiguration.gearOutCamOut.jerk := -1.0;
   cmCathodeMainPnP1AxisY.commandConfiguration.gearOutCamOut.syncOutDirection := 3;
   cmCathodeMainPnP1AxisY.commandConfiguration.gearOutCamOut.gearOutCamOutMode := -1;
   cmCathodeMainPnP1AxisY.commandConfiguration.phasing.phaseShift := 0.0;
   cmCathodeMainPnP1AxisY.commandConfiguration.phasing.velocity := -1.0;
   cmCathodeMainPnP1AxisY.commandConfiguration.phasing.acceleration := -1.0;
   cmCathodeMainPnP1AxisY.commandConfiguration.phasing.deceleration := -1.0;
   cmCathodeMainPnP1AxisY.commandConfiguration.phasing.jerk := -1.0;
   cmCathodeMainPnP1AxisY.commandConfiguration.phasing.profileReference := 0;
   cmCathodeMainPnP1AxisY.commandConfiguration.phasing.phasingDistance := 0.0;
   cmCathodeMainPnP1AxisY.commandConfiguration.phasing.startPosition := 0.0;
   cmCathodeMainPnP1AxisY.commandConfiguration.phasing.direction := 3;
   cmCathodeMainPnP1AxisY.commandConfiguration.phasing.phaseAbsolute := TRUE;
   cmCathodeMainPnP1AxisY.commandConfiguration.phasing.phaseShiftChangeOnTheFly := FALSE;
   cmCathodeMainPnP1AxisY.commandConfiguration.offset.offset := 0.0;
   cmCathodeMainPnP1AxisY.commandConfiguration.offset.profileReference := 1;
   cmCathodeMainPnP1AxisY.commandConfiguration.offset.offsetDistance := 0.0;
   cmCathodeMainPnP1AxisY.commandConfiguration.offset.startPosition := 0.0;
   cmCathodeMainPnP1AxisY.commandConfiguration.offset.direction := 3;
   cmCathodeMainPnP1AxisY.commandConfiguration.offset.offsetAbsolute := TRUE;
   cmCathodeMainPnP1AxisY.commandConfiguration.offset.offsetChangeOnTheFly := FALSE;
   cmCathodeMainPnP1AxisY.commands.enableAxis := FALSE;
   cmCathodeMainPnP1AxisY.commands.resetAxis := FALSE;
   cmCathodeMainPnP1AxisY.commands.openBrake := FALSE;
   cmCathodeMainPnP1AxisY.commands.jogForward := FALSE;
   cmCathodeMainPnP1AxisY.commands.jogBackward := FALSE;
   cmCathodeMainPnP1AxisY.commands.moveVelocity := FALSE;
   cmCathodeMainPnP1AxisY.commands.stop := FALSE;
   cmCathodeMainPnP1AxisY.commands.fastStop := FALSE;
   cmCathodeMainPnP1AxisY.commands.torqueLimiting := FALSE;
   cmCathodeMainPnP1AxisY.commands.homing := FALSE;
   cmCathodeMainPnP1AxisY.commands.posRelative := FALSE;
   cmCathodeMainPnP1AxisY.commands.posAbsolute := FALSE;
   cmCathodeMainPnP1AxisY.commands.posSuperimposed := FALSE;
   cmCathodeMainPnP1AxisY.commands.haltSuperimposed := FALSE;
   cmCathodeMainPnP1AxisY.commands.selectSetPosition := -1;
   cmCathodeMainPnP1AxisY.commands.reset := FALSE;
   cmCathodeMainPnP1AxisY.monitoring.valid := FALSE;
   cmCathodeMainPnP1AxisY.monitoring.busy := TRUE;
   cmCathodeMainPnP1AxisY.monitoring.error := TRUE;
   cmCathodeMainPnP1AxisY.monitoring.status := 16#8600;
   cmCathodeMainPnP1AxisY.monitoring.subfunctionStatus := 16#8001;
   cmCathodeMainPnP1AxisY.monitoring.axisEnabled := FALSE;
   cmCathodeMainPnP1AxisY.monitoring.resetActive := FALSE;
   cmCathodeMainPnP1AxisY.monitoring.inVelocity := FALSE;
   cmCathodeMainPnP1AxisY.monitoring.inLimitation := FALSE;
   cmCathodeMainPnP1AxisY.monitoring.inClamping := FALSE;
   cmCathodeMainPnP1AxisY.monitoring.startSync := FALSE;
   cmCathodeMainPnP1AxisY.monitoring.inSync := FALSE;
   cmCathodeMainPnP1AxisY.monitoring.inSimulation := FALSE;
   cmCathodeMainPnP1AxisY.monitoring.jogSelected := FALSE;
   cmCathodeMainPnP1AxisY.monitoring.moveVelocitySelected := FALSE;
   cmCathodeMainPnP1AxisY.monitoring.stopSelected := FALSE;
   cmCathodeMainPnP1AxisY.monitoring.fastStopSelected := FALSE;
   cmCathodeMainPnP1AxisY.monitoring.torqueLimitingSelected := FALSE;
   cmCathodeMainPnP1AxisY.monitoring.homingSelected := FALSE;
   cmCathodeMainPnP1AxisY.monitoring.posRelativeSelected := FALSE;
   cmCathodeMainPnP1AxisY.monitoring.posAbsoluteSelected := FALSE;
   cmCathodeMainPnP1AxisY.monitoring.posSuperimposedSelected := FALSE;
   cmCathodeMainPnP1AxisY.monitoring.haltSuperimposedSelected := FALSE;
   cmCathodeMainPnP1AxisY.monitoring.commandBusy := FALSE;
   cmCathodeMainPnP1AxisY.monitoring.commandDone := FALSE;
   cmCathodeMainPnP1AxisY.monitoring.commandAborted := FALSE;
   cmCathodeMainPnP1AxisY.monitoring.homingCommandBusy := FALSE;
   cmCathodeMainPnP1AxisY.monitoring.homingCommandDone := FALSE;
   cmCathodeMainPnP1AxisY.monitoring.homingCommandAborted := FALSE;
   cmCathodeMainPnP1AxisY.monitoring.superimposedBusy := FALSE;
   cmCathodeMainPnP1AxisY.monitoring.superimposedDone := FALSE;
   cmCathodeMainPnP1AxisY.monitoring.superimposedAborted := FALSE;
   cmCathodeMainPnP1AxisY.monitoring.actualPosition := 0.0;
   cmCathodeMainPnP1AxisY.monitoring.actualSpeed := 0.0;
   cmCathodeMainPnP1AxisY.monitoring.speedUnit := 1062;
   cmCathodeMainPnP1AxisY.monitoring.positionUnit := 1013;
   cmCathodeMainPnP1AxisY.monitoring.axisType := 1;
   cmCathodeMainPnP1AxisY.monitoring.interlockGeneralOut := TRUE;
   cmCathodeMainPnP1AxisY.monitoring.interlockJogForwardOut := TRUE;
   cmCathodeMainPnP1AxisY.monitoring.interlockJogBackwardOut := TRUE;
   cmCathodeMainPnP1AxisZ.commandConfiguration.generalSettings.stopOnError := TRUE;
   cmCathodeMainPnP1AxisZ.commandConfiguration.generalSettings.resetWithRestart := FALSE;
   cmCathodeMainPnP1AxisZ.commandConfiguration.generalSettings.abortWaitingSyncCmd := TRUE;
   cmCathodeMainPnP1AxisZ.commandConfiguration.power.startMode := 1;
   cmCathodeMainPnP1AxisZ.commandConfiguration.power.stopMode := 0;
   cmCathodeMainPnP1AxisZ.commandConfiguration.power.syncMotionSimulation := FALSE;
   cmCathodeMainPnP1AxisZ.commandConfiguration.power.syncMotionSimulationExtendedMode := -1;
   cmCathodeMainPnP1AxisZ.commandConfiguration.jog.velocity := 10.0;
   cmCathodeMainPnP1AxisZ.commandConfiguration.jog.acceleration := -1.0;
   cmCathodeMainPnP1AxisZ.commandConfiguration.jog.deceleration := -1.0;
   cmCathodeMainPnP1AxisZ.commandConfiguration.jog.jerk := -1.0;
   cmCathodeMainPnP1AxisZ.commandConfiguration.jog.positionControlled := TRUE;
   cmCathodeMainPnP1AxisZ.commandConfiguration.jog.increment := 0.0;
   cmCathodeMainPnP1AxisZ.commandConfiguration.jog.mode := 0;
   cmCathodeMainPnP1AxisZ.commandConfiguration.moveVelocity.velocity := 0.0;
   cmCathodeMainPnP1AxisZ.commandConfiguration.moveVelocity.acceleration := -1.0;
   cmCathodeMainPnP1AxisZ.commandConfiguration.moveVelocity.deceleration := -1.0;
   cmCathodeMainPnP1AxisZ.commandConfiguration.moveVelocity.jerk := -1.0;
   cmCathodeMainPnP1AxisZ.commandConfiguration.moveVelocity.direction := 0;
   cmCathodeMainPnP1AxisZ.commandConfiguration.moveVelocity.positionControlled := TRUE;
   cmCathodeMainPnP1AxisZ.commandConfiguration.moveVelocity.velocityChangeOnTheFly := FALSE;
   cmCathodeMainPnP1AxisZ.commandConfiguration.stop.deceleration := -1.0;
   cmCathodeMainPnP1AxisZ.commandConfiguration.stop.jerk := -1.0;
   cmCathodeMainPnP1AxisZ.commandConfiguration.stop.abortAcceleration := FALSE;
   cmCathodeMainPnP1AxisZ.commandConfiguration.fastStop.deceleration := -1.0;
   cmCathodeMainPnP1AxisZ.commandConfiguration.fastStop.jerk := -1.0;
   cmCathodeMainPnP1AxisZ.commandConfiguration.fastStop.abortAcceleration := FALSE;
   cmCathodeMainPnP1AxisZ.commandConfiguration.fastStop.replaceStopPossible := FALSE;
   cmCathodeMainPnP1AxisZ.commandConfiguration.torqueLimiting.limit := -1.0;
   cmCathodeMainPnP1AxisZ.commandConfiguration.torqueLimiting.mode := 0;
   cmCathodeMainPnP1AxisZ.commandConfiguration.homing.position := 0.0;
   cmCathodeMainPnP1AxisZ.commandConfiguration.homing.mode := 0;
   cmCathodeMainPnP1AxisZ.commandConfiguration.homing.sensor := 0;
   cmCathodeMainPnP1AxisZ.commandConfiguration.homing.extendedMode := -1;
   cmCathodeMainPnP1AxisZ.commandConfiguration.homing.extendedModeTorqueLimit := 0.0;
   cmCathodeMainPnP1AxisZ.commandConfiguration.homing.extendedModeTargetPosition := 0.0;
   cmCathodeMainPnP1AxisZ.commandConfiguration.posRelative.distance := 0.0;
   cmCathodeMainPnP1AxisZ.commandConfiguration.posRelative.velocity := -1.0;
   cmCathodeMainPnP1AxisZ.commandConfiguration.posRelative.acceleration := -1.0;
   cmCathodeMainPnP1AxisZ.commandConfiguration.posRelative.deceleration := -1.0;
   cmCathodeMainPnP1AxisZ.commandConfiguration.posRelative.jerk := -1.0;
   cmCathodeMainPnP1AxisZ.commandConfiguration.posRelative.direction := 0;
   cmCathodeMainPnP1AxisZ.commandConfiguration.posAbsolute.position := 0.0;
   cmCathodeMainPnP1AxisZ.commandConfiguration.posAbsolute.velocity := -1.0;
   cmCathodeMainPnP1AxisZ.commandConfiguration.posAbsolute.acceleration := -1.0;
   cmCathodeMainPnP1AxisZ.commandConfiguration.posAbsolute.deceleration := -1.0;
   cmCathodeMainPnP1AxisZ.commandConfiguration.posAbsolute.jerk := -1.0;
   cmCathodeMainPnP1AxisZ.commandConfiguration.posAbsolute.direction := 1;
   cmCathodeMainPnP1AxisZ.commandConfiguration.posAbsolute.positionChangeOnTheFly := FALSE;
   cmCathodeMainPnP1AxisZ.commandConfiguration.posAbsolute.velocityChangeOnTheFly := FALSE;
   cmCathodeMainPnP1AxisZ.commandConfiguration.posSuperimposed.distance := 0.0;
   cmCathodeMainPnP1AxisZ.commandConfiguration.posSuperimposed.velocityDiff := -1.0;
   cmCathodeMainPnP1AxisZ.commandConfiguration.posSuperimposed.acceleration := -1.0;
   cmCathodeMainPnP1AxisZ.commandConfiguration.posSuperimposed.deceleration := -1.0;
   cmCathodeMainPnP1AxisZ.commandConfiguration.posSuperimposed.jerk := -1.0;
   cmCathodeMainPnP1AxisZ.commandConfiguration.posSuperimposed.direction := 0;
   cmCathodeMainPnP1AxisZ.commandConfiguration.haltSuperimposed.deceleration := -1.0;
   cmCathodeMainPnP1AxisZ.commandConfiguration.haltSuperimposed.jerk := -1.0;
   cmCathodeMainPnP1AxisZ.commandConfiguration.haltSuperimposed.abortAcceleration := FALSE;
   cmCathodeMainPnP1AxisZ.commandConfiguration.gearInRelative.ratioNumerator := 1;
   cmCathodeMainPnP1AxisZ.commandConfiguration.gearInRelative.ratioDenominator := 1;
   cmCathodeMainPnP1AxisZ.commandConfiguration.gearInRelative.acceleration := -1.0;
   cmCathodeMainPnP1AxisZ.commandConfiguration.gearInRelative.deceleration := -1.0;
   cmCathodeMainPnP1AxisZ.commandConfiguration.gearInRelative.jerk := -1.0;
   cmCathodeMainPnP1AxisZ.commandConfiguration.gearInRelative.ratioChangeOnTheFly := FALSE;
   cmCathodeMainPnP1AxisZ.commandConfiguration.gearInAbsolute.ratioNumerator := 1;
   cmCathodeMainPnP1AxisZ.commandConfiguration.gearInAbsolute.ratioDenominator := 1;
   cmCathodeMainPnP1AxisZ.commandConfiguration.gearInAbsolute.masterSyncPosition := 0.0;
   cmCathodeMainPnP1AxisZ.commandConfiguration.gearInAbsolute.slaveSyncPosition := 0.0;
   cmCathodeMainPnP1AxisZ.commandConfiguration.gearInAbsolute.syncProfileReference := 1;
   cmCathodeMainPnP1AxisZ.commandConfiguration.gearInAbsolute.masterStartDistance := 0.0;
   cmCathodeMainPnP1AxisZ.commandConfiguration.gearInAbsolute.velocity := -1.0;
   cmCathodeMainPnP1AxisZ.commandConfiguration.gearInAbsolute.acceleration := -1.0;
   cmCathodeMainPnP1AxisZ.commandConfiguration.gearInAbsolute.deceleration := -1.0;
   cmCathodeMainPnP1AxisZ.commandConfiguration.gearInAbsolute.jerk := -1.0;
   cmCathodeMainPnP1AxisZ.commandConfiguration.gearInAbsolute.syncDirection := 1;
   cmCathodeMainPnP1AxisZ.commandConfiguration.gearInAbsolute.ratioChangeOnTheFly := FALSE;
   cmCathodeMainPnP1AxisZ.commandConfiguration.gearInVelocity.continuousUpdate := FALSE;
   cmCathodeMainPnP1AxisZ.commandConfiguration.gearInVelocity.ratioNumerator := 1;
   cmCathodeMainPnP1AxisZ.commandConfiguration.gearInVelocity.ratioDenominator := 1;
   cmCathodeMainPnP1AxisZ.commandConfiguration.gearInVelocity.acceleration := -1.0;
   cmCathodeMainPnP1AxisZ.commandConfiguration.gearInVelocity.deceleration := -1.0;
   cmCathodeMainPnP1AxisZ.commandConfiguration.gearInVelocity.jerk := -1.0;
   cmCathodeMainPnP1AxisZ.commandConfiguration.gearInVelocity.positionControlled := FALSE;
   cmCathodeMainPnP1AxisZ.commandConfiguration.camIn.masterOffset := 0.0;
   cmCathodeMainPnP1AxisZ.commandConfiguration.camIn.slaveOffset := 0.0;
   cmCathodeMainPnP1AxisZ.commandConfiguration.camIn.masterScaling := 1.0;
   cmCathodeMainPnP1AxisZ.commandConfiguration.camIn.slaveScaling := 1.0;
   cmCathodeMainPnP1AxisZ.commandConfiguration.camIn.masterSyncPosition := 0.0;
   cmCathodeMainPnP1AxisZ.commandConfiguration.camIn.syncProfileReference := 1;
   cmCathodeMainPnP1AxisZ.commandConfiguration.camIn.masterStartDistance := 0.0;
   cmCathodeMainPnP1AxisZ.commandConfiguration.camIn.velocity := -1.0;
   cmCathodeMainPnP1AxisZ.commandConfiguration.camIn.acceleration := -1.0;
   cmCathodeMainPnP1AxisZ.commandConfiguration.camIn.deceleration := -1.0;
   cmCathodeMainPnP1AxisZ.commandConfiguration.camIn.jerk := -1.0;
   cmCathodeMainPnP1AxisZ.commandConfiguration.camIn.applicationMode := 0;
   cmCathodeMainPnP1AxisZ.commandConfiguration.camIn.syncDirection := 1;
   cmCathodeMainPnP1AxisZ.commandConfiguration.gearOutCamOut.slavePosition := 0.0;
   cmCathodeMainPnP1AxisZ.commandConfiguration.gearOutCamOut.syncProfileReference := 1;
   cmCathodeMainPnP1AxisZ.commandConfiguration.gearOutCamOut.masterStopDistance := 0.0;
   cmCathodeMainPnP1AxisZ.commandConfiguration.gearOutCamOut.deceleration := -1.0;
   cmCathodeMainPnP1AxisZ.commandConfiguration.gearOutCamOut.jerk := -1.0;
   cmCathodeMainPnP1AxisZ.commandConfiguration.gearOutCamOut.syncOutDirection := 3;
   cmCathodeMainPnP1AxisZ.commandConfiguration.gearOutCamOut.gearOutCamOutMode := -1;
   cmCathodeMainPnP1AxisZ.commandConfiguration.phasing.phaseShift := 0.0;
   cmCathodeMainPnP1AxisZ.commandConfiguration.phasing.velocity := -1.0;
   cmCathodeMainPnP1AxisZ.commandConfiguration.phasing.acceleration := -1.0;
   cmCathodeMainPnP1AxisZ.commandConfiguration.phasing.deceleration := -1.0;
   cmCathodeMainPnP1AxisZ.commandConfiguration.phasing.jerk := -1.0;
   cmCathodeMainPnP1AxisZ.commandConfiguration.phasing.profileReference := 0;
   cmCathodeMainPnP1AxisZ.commandConfiguration.phasing.phasingDistance := 0.0;
   cmCathodeMainPnP1AxisZ.commandConfiguration.phasing.startPosition := 0.0;
   cmCathodeMainPnP1AxisZ.commandConfiguration.phasing.direction := 3;
   cmCathodeMainPnP1AxisZ.commandConfiguration.phasing.phaseAbsolute := TRUE;
   cmCathodeMainPnP1AxisZ.commandConfiguration.phasing.phaseShiftChangeOnTheFly := FALSE;
   cmCathodeMainPnP1AxisZ.commandConfiguration.offset.offset := 0.0;
   cmCathodeMainPnP1AxisZ.commandConfiguration.offset.profileReference := 1;
   cmCathodeMainPnP1AxisZ.commandConfiguration.offset.offsetDistance := 0.0;
   cmCathodeMainPnP1AxisZ.commandConfiguration.offset.startPosition := 0.0;
   cmCathodeMainPnP1AxisZ.commandConfiguration.offset.direction := 3;
   cmCathodeMainPnP1AxisZ.commandConfiguration.offset.offsetAbsolute := TRUE;
   cmCathodeMainPnP1AxisZ.commandConfiguration.offset.offsetChangeOnTheFly := FALSE;
   cmCathodeMainPnP1AxisZ.commands.enableAxis := FALSE;
   cmCathodeMainPnP1AxisZ.commands.resetAxis := FALSE;
   cmCathodeMainPnP1AxisZ.commands.openBrake := FALSE;
   cmCathodeMainPnP1AxisZ.commands.jogForward := FALSE;
   cmCathodeMainPnP1AxisZ.commands.jogBackward := FALSE;
   cmCathodeMainPnP1AxisZ.commands.moveVelocity := FALSE;
   cmCathodeMainPnP1AxisZ.commands.stop := FALSE;
   cmCathodeMainPnP1AxisZ.commands.fastStop := FALSE;
   cmCathodeMainPnP1AxisZ.commands.torqueLimiting := FALSE;
   cmCathodeMainPnP1AxisZ.commands.homing := FALSE;
   cmCathodeMainPnP1AxisZ.commands.posRelative := FALSE;
   cmCathodeMainPnP1AxisZ.commands.posAbsolute := FALSE;
   cmCathodeMainPnP1AxisZ.commands.posSuperimposed := FALSE;
   cmCathodeMainPnP1AxisZ.commands.haltSuperimposed := FALSE;
   cmCathodeMainPnP1AxisZ.commands.selectSetPosition := -1;
   cmCathodeMainPnP1AxisZ.commands.reset := FALSE;
   cmCathodeMainPnP1AxisZ.monitoring.valid := FALSE;
   cmCathodeMainPnP1AxisZ.monitoring.busy := TRUE;
   cmCathodeMainPnP1AxisZ.monitoring.error := TRUE;
   cmCathodeMainPnP1AxisZ.monitoring.status := 16#8600;
   cmCathodeMainPnP1AxisZ.monitoring.subfunctionStatus := 16#8001;
   cmCathodeMainPnP1AxisZ.monitoring.axisEnabled := FALSE;
   cmCathodeMainPnP1AxisZ.monitoring.resetActive := FALSE;
   cmCathodeMainPnP1AxisZ.monitoring.inVelocity := FALSE;
   cmCathodeMainPnP1AxisZ.monitoring.inLimitation := FALSE;
   cmCathodeMainPnP1AxisZ.monitoring.inClamping := FALSE;
   cmCathodeMainPnP1AxisZ.monitoring.startSync := FALSE;
   cmCathodeMainPnP1AxisZ.monitoring.inSync := FALSE;
   cmCathodeMainPnP1AxisZ.monitoring.inSimulation := FALSE;
   cmCathodeMainPnP1AxisZ.monitoring.jogSelected := FALSE;
   cmCathodeMainPnP1AxisZ.monitoring.moveVelocitySelected := FALSE;
   cmCathodeMainPnP1AxisZ.monitoring.stopSelected := FALSE;
   cmCathodeMainPnP1AxisZ.monitoring.fastStopSelected := FALSE;
   cmCathodeMainPnP1AxisZ.monitoring.torqueLimitingSelected := FALSE;
   cmCathodeMainPnP1AxisZ.monitoring.homingSelected := FALSE;
   cmCathodeMainPnP1AxisZ.monitoring.posRelativeSelected := FALSE;
   cmCathodeMainPnP1AxisZ.monitoring.posAbsoluteSelected := FALSE;
   cmCathodeMainPnP1AxisZ.monitoring.posSuperimposedSelected := FALSE;
   cmCathodeMainPnP1AxisZ.monitoring.haltSuperimposedSelected := FALSE;
   cmCathodeMainPnP1AxisZ.monitoring.commandBusy := FALSE;
   cmCathodeMainPnP1AxisZ.monitoring.commandDone := FALSE;
   cmCathodeMainPnP1AxisZ.monitoring.commandAborted := FALSE;
   cmCathodeMainPnP1AxisZ.monitoring.homingCommandBusy := FALSE;
   cmCathodeMainPnP1AxisZ.monitoring.homingCommandDone := FALSE;
   cmCathodeMainPnP1AxisZ.monitoring.homingCommandAborted := FALSE;
   cmCathodeMainPnP1AxisZ.monitoring.superimposedBusy := FALSE;
   cmCathodeMainPnP1AxisZ.monitoring.superimposedDone := FALSE;
   cmCathodeMainPnP1AxisZ.monitoring.superimposedAborted := FALSE;
   cmCathodeMainPnP1AxisZ.monitoring.actualPosition := 5.609;
   cmCathodeMainPnP1AxisZ.monitoring.actualSpeed := 0.0;
   cmCathodeMainPnP1AxisZ.monitoring.speedUnit := 1062;
   cmCathodeMainPnP1AxisZ.monitoring.positionUnit := 1013;
   cmCathodeMainPnP1AxisZ.monitoring.axisType := 1;
   cmCathodeMainPnP1AxisZ.monitoring.interlockGeneralOut := TRUE;
   cmCathodeMainPnP1AxisZ.monitoring.interlockJogForwardOut := TRUE;
   cmCathodeMainPnP1AxisZ.monitoring.interlockJogBackwardOut := TRUE;
   cmCathodeMainPnP2AxisZ.commandConfiguration.generalSettings.stopOnError := TRUE;
   cmCathodeMainPnP2AxisZ.commandConfiguration.generalSettings.resetWithRestart := FALSE;
   cmCathodeMainPnP2AxisZ.commandConfiguration.generalSettings.abortWaitingSyncCmd := TRUE;
   cmCathodeMainPnP2AxisZ.commandConfiguration.power.startMode := 1;
   cmCathodeMainPnP2AxisZ.commandConfiguration.power.stopMode := 0;
   cmCathodeMainPnP2AxisZ.commandConfiguration.power.syncMotionSimulation := FALSE;
   cmCathodeMainPnP2AxisZ.commandConfiguration.power.syncMotionSimulationExtendedMode := -1;
   cmCathodeMainPnP2AxisZ.commandConfiguration.jog.velocity := 10.0;
   cmCathodeMainPnP2AxisZ.commandConfiguration.jog.acceleration := -1.0;
   cmCathodeMainPnP2AxisZ.commandConfiguration.jog.deceleration := -1.0;
   cmCathodeMainPnP2AxisZ.commandConfiguration.jog.jerk := -1.0;
   cmCathodeMainPnP2AxisZ.commandConfiguration.jog.positionControlled := TRUE;
   cmCathodeMainPnP2AxisZ.commandConfiguration.jog.increment := 0.0;
   cmCathodeMainPnP2AxisZ.commandConfiguration.jog.mode := 0;
